C01824=1116.174,356.442,-84.946,-177.177,11.022,149.491
C01825=1116.170,356.689,-84.982,-177.174,11.024,149.491
C01826=1116.166,356.936,-85.017,-177.170,11.027,149.490
C01827=1116.163,357.184,-85.053,-177.167,11.029,149.490
C01828=1116.158,357.431,-85.089,-177.163,11.031,149.490
C01829=1116.155,357.678,-85.125,-177.160,11.034,149.490
C01830=1116.151,357.926,-85.161,-177.157,11.036,149.489
C01831=1116.147,358.173,-85.196,-177.153,11.039,149.489
C01832=1116.143,358.421,-85.232,-177.150,11.041,149.489
C01833=1116.140,358.668,-85.269,-177.146,11.043,149.489
C01834=1116.136,358.916,-85.304,-177.143,11.046,149.488
C01835=1116.132,359.163,-85.340,-177.140,11.048,149.488
C01836=1116.128,359.411,-85.376,-177.136,11.051,149.488
C01837=1116.125,359.658,-85.412,-177.133,11.053,149.487
C01838=1116.121,359.905,-85.448,-177.129,11.055,149.487
C01839=1116.117,360.153,-85.484,-177.126,11.058,149.487
C01840=1116.113,360.400,-85.520,-177.123,11.060,149.487
C01841=1116.110,360.647,-85.556,-177.119,11.063,149.486
C01842=1116.105,360.895,-85.593,-177.116,11.065,149.486
C01843=1116.102,361.142,-85.628,-177.113,11.067,149.486
C01844=1116.098,361.390,-85.664,-177.109,11.070,149.486
C01845=1116.094,361.602,-85.695,-177.107,11.072,149.486
C01846=1116.091,361.813,-85.726,-177.104,11.073,149.485
C01847=1116.089,362.025,-85.757,-177.101,11.076,149.485
C01848=1116.085,362.237,-85.788,-177.098,11.077,149.485
C01849=1116.082,362.449,-85.819,-177.095,11.080,149.485
C01850=1116.078,362.662,-85.850,-177.092,11.082,149.484
C01851=1116.075,362.874,-85.881,-177.090,11.084,149.484
C01852=1116.072,363.085,-85.911,-177.086,11.086,149.484
C01853=1116.068,363.332,-85.948,-177.083,11.088,149.484
C01854=1116.064,363.579,-85.984,-177.079,11.091,149.483
C01855=1116.061,363.828,-86.021,-177.076,11.093,149.483
C01856=1116.057,364.075,-86.057,-177.073,11.096,149.483
C01857=1116.054,364.322,-86.093,-177.069,11.098,149.483
C01858=1116.050,364.569,-86.129,-177.066,11.100,149.482
C01859=1116.046,364.816,-86.166,-177.062,11.103,149.482
C01860=1116.042,365.064,-86.202,-177.059,11.105,149.482
C01861=1116.038,365.311,-86.238,-177.056,11.108,149.482
C01862=1116.034,365.559,-86.274,-177.052,11.110,149.482
C01863=1116.030,365.806,-86.311,-177.049,11.112,149.481
C01864=1116.027,366.053,-86.347,-177.046,11.114,149.481
C01865=1116.022,366.300,-86.384,-177.043,11.116,149.481
C01866=1116.019,366.548,-86.420,-177.040,11.119,149.480
C01867=1116.015,366.795,-86.457,-177.036,11.121,149.480
C01868=1116.012,367.042,-86.493,-177.033,11.124,149.480
C01869=1116.008,367.290,-86.530,-177.029,11.126,149.480
C01870=1116.003,367.537,-86.566,-177.026,11.129,149.479
C01871=1116.000,367.784,-86.603,-177.023,11.131,149.479
C01872=1115.996,368.031,-86.639,-177.019,11.133,149.479
C01873=1115.993,368.278,-86.676,-177.016,11.136,149.479
C01874=1115.989,368.526,-86.713,-177.013,11.138,149.479
C01875=1115.985,368.773,-86.750,-177.009,11.141,149.478
C01876=1115.981,369.021,-86.785,-177.006,11.143,149.478
C01877=1115.977,369.268,-86.822,-177.002,11.146,149.478
C01878=1115.973,369.515,-86.859,-176.999,11.148,149.478
C01879=1115.970,369.762,-86.895,-176.996,11.150,149.477
C01880=1115.966,370.010,-86.932,-176.993,11.153,149.477
C01881=1115.962,370.257,-86.969,-176.989,11.155,149.477
C01882=1115.959,370.504,-87.006,-176.987,11.157,149.477
C01883=1115.955,370.751,-87.042,-176.983,11.160,149.477
C01884=1115.951,370.999,-87.079,-176.980,11.162,149.476
C01885=1115.948,371.246,-87.116,-176.977,11.165,149.476
C01886=1115.944,371.493,-87.153,-176.973,11.167,149.476
C01887=1115.940,371.740,-87.190,-176.970,11.170,149.476
C01888=1115.936,371.988,-87.227,-176.966,11.172,149.475
C01889=1115.933,372.235,-87.263,-176.963,11.174,149.475
C01890=1115.929,372.482,-87.300,-176.960,11.177,149.475
C01891=1115.925,372.730,-87.337,-176.956,11.179,149.475
C01892=1115.921,372.977,-87.374,-176.953,11.182,149.474
C01893=1115.918,373.224,-87.411,-176.950,11.184,149.474
C01894=1115.914,373.471,-87.448,-176.947,11.187,149.474
C01895=1115.910,373.718,-87.485,-176.943,11.189,149.474
C01896=1115.906,373.965,-87.522,-176.940,11.192,149.474
C01897=1115.902,374.213,-87.559,-176.937,11.194,149.473
C01898=1115.898,374.460,-87.596,-176.934,11.197,149.473
C01899=1115.895,374.707,-87.633,-176.930,11.199,149.473
C01900=1115.892,374.955,-87.670,-176.928,11.201,149.473
C01901=1115.888,375.166,-87.702,-176.925,11.203,149.473
C01902=1115.885,375.379,-87.733,-176.922,11.205,149.473
C01903=1115.881,375.590,-87.765,-176.919,11.208,149.473
C01904=1115.879,375.802,-87.797,-176.916,11.210,149.472
C01905=1115.875,376.014,-87.829,-176.914,11.211,149.472
C01906=1115.873,376.226,-87.861,-176.911,11.214,149.472
C01907=1115.868,376.437,-87.893,-176.908,11.216,149.472
C01908=1115.866,376.649,-87.925,-176.905,11.219,149.472
C01909=1115.862,376.896,-87.962,-176.902,11.221,149.472
C01910=1115.858,377.144,-87.999,-176.899,11.223,149.471
C01911=1115.854,377.391,-88.037,-176.896,11.225,149.471
C01912=1115.851,377.638,-88.073,-176.893,11.228,149.471
C01913=1115.847,377.886,-88.110,-176.890,11.231,149.471
C01914=1115.844,378.132,-88.148,-176.886,11.233,149.471
C01915=1115.840,378.379,-88.184,-176.883,11.236,149.471
C01916=1115.836,378.627,-88.222,-176.880,11.238,149.470
C01917=1115.832,378.874,-88.259,-176.877,11.241,149.470
C01918=1115.829,379.120,-88.297,-176.874,11.243,149.470
C01919=1115.825,379.368,-88.334,-176.870,11.246,149.470
C01920=1115.821,379.615,-88.372,-176.867,11.248,149.470
C01921=1115.818,379.863,-88.409,-176.864,11.251,149.470
C01922=1115.814,380.109,-88.446,-176.861,11.254,149.470
C01923=1115.809,380.357,-88.484,-176.858,11.256,149.469
C01924=1115.806,380.604,-88.522,-176.855,11.259,149.469
C01925=1115.802,380.851,-88.559,-176.851,11.261,149.469
C01926=1115.799,381.099,-88.597,-176.848,11.264,149.469
C01927=1115.795,381.345,-88.634,-176.845,11.267,149.469
C01928=1115.791,381.593,-88.671,-176.842,11.269,149.469
C01929=1115.788,381.840,-88.709,-176.839,11.272,149.469
C01930=1115.784,382.087,-88.746,-176.836,11.275,149.468
C01931=1115.780,382.334,-88.784,-176.832,11.277,149.468
C01932=1115.777,382.581,-88.821,-176.829,11.280,149.468
C01933=1115.773,382.829,-88.859,-176.826,11.282,149.468
C01934=1115.769,383.075,-88.897,-176.823,11.285,149.468
C01935=1115.765,383.323,-88.935,-176.820,11.288,149.468
C01936=1115.762,383.569,-88.972,-176.817,11.290,149.468
C01937=1115.758,383.817,-89.009,-176.815,11.293,149.468
C01938=1115.754,384.064,-89.047,-176.813,11.295,149.468
C01939=1115.751,384.311,-89.085,-176.810,11.298,149.468
C01940=1115.747,384.558,-89.123,-176.808,11.300,149.468
C01941=1115.743,384.805,-89.161,-176.806,11.302,149.468
C01942=1115.739,385.052,-89.198,-176.803,11.305,149.468
C01943=1115.736,385.300,-89.236,-176.801,11.307,149.468
C01944=1115.732,385.546,-89.273,-176.798,11.309,149.468
C01945=1115.729,385.793,-89.311,-176.796,11.312,149.468
C01946=1115.725,386.040,-89.350,-176.794,11.314,149.468
C01947=1115.721,386.288,-89.388,-176.791,11.317,149.468
C01948=1115.717,386.535,-89.424,-176.789,11.319,149.468
C01949=1115.714,386.782,-89.462,-176.787,11.321,149.468
C01950=1115.710,387.030,-89.501,-176.784,11.324,149.468
C01951=1115.706,387.276,-89.538,-176.782,11.327,149.468
C01952=1115.703,387.523,-89.576,-176.779,11.330,149.468
C01953=1115.699,387.770,-89.614,-176.778,11.332,149.469
C01954=1115.695,388.018,-89.652,-176.775,11.335,149.469
C01955=1115.692,388.264,-89.690,-176.773,11.337,149.469
C01956=1115.689,388.511,-89.728,-176.770,11.340,149.469
C01957=1115.685,388.724,-89.761,-176.768,11.343,149.469
C01958=1115.682,388.934,-89.793,-176.767,11.345,149.469
C01959=1115.679,389.147,-89.826,-176.765,11.347,149.469
C01960=1115.676,389.358,-89.858,-176.763,11.350,149.469
C01961=1115.673,389.571,-89.891,-176.761,11.352,149.470
C01962=1115.670,389.781,-89.923,-176.759,11.355,149.470
C01963=1115.666,389.994,-89.956,-176.757,11.357,149.470
C01964=1115.664,390.205,-89.988,-176.755,11.359,149.470
C01965=1115.660,390.453,-90.027,-176.753,11.362,149.470
C01966=1115.656,390.699,-90.065,-176.750,11.366,149.470
C01967=1115.653,390.946,-90.102,-176.748,11.368,149.470
C01968=1115.648,391.193,-90.141,-176.746,11.371,149.471
C01969=1115.645,391.441,-90.179,-176.744,11.375,149.471
C01970=1115.642,391.688,-90.217,-176.742,11.377,149.471
C01971=1115.638,391.934,-90.255,-176.739,11.380,149.471
C01972=1115.634,392.181,-90.293,-176.737,11.383,149.472
C01973=1115.631,392.429,-90.332,-176.735,11.386,149.472
C01974=1115.627,392.676,-90.369,-176.733,11.389,149.472
C01975=1115.624,392.923,-90.407,-176.731,11.392,149.472
C01976=1115.620,393.170,-90.447,-176.729,11.396,149.473
C01977=1115.616,393.416,-90.484,-176.726,11.399,149.473
C01978=1115.612,393.664,-90.523,-176.725,11.402,149.473
C01979=1115.609,393.911,-90.561,-176.723,11.405,149.474
C01980=1115.605,394.158,-90.599,-176.720,11.408,149.474
C01981=1115.602,394.405,-90.638,-176.718,11.412,149.474
C01982=1115.598,394.652,-90.676,-176.716,11.415,149.475
C01983=1115.594,394.899,-90.714,-176.714,11.419,149.475
C01984=1115.590,395.146,-90.753,-176.712,11.421,149.475
C01985=1115.587,395.393,-90.791,-176.710,11.425,149.476
C01986=1115.583,395.640,-90.829,-176.708,11.428,149.476
C01987=1115.580,395.887,-90.868,-176.706,11.432,149.476
C01988=1115.576,396.134,-90.906,-176.704,11.435,149.477
C01989=1115.573,396.381,-90.944,-176.702,11.439,149.477
C01990=1115.568,396.628,-90.983,-176.700,11.443,149.478
C01991=1115.565,396.875,-91.021,-176.698,11.446,149.478
C01992=1115.562,397.122,-91.060,-176.696,11.450,149.478
C01993=1115.558,397.369,-91.098,-176.694,11.453,149.479
C01994=1115.554,397.616,-91.136,-176.692,11.457,149.479
C01995=1115.551,397.863,-91.175,-176.690,11.461,149.480
C01996=1115.547,398.110,-91.214,-176.688,11.464,149.480
C01997=1115.543,398.357,-91.252,-176.686,11.468,149.481
C01998=1115.540,398.604,-91.290,-176.684,11.471,149.481
C01999=1115.536,398.851,-91.330,-176.683,11.475,149.482
C02000=1115.533,399.098,-91.368,-176.680,11.480,149.482
C02001=1115.529,399.344,-91.406,-176.678,11.483,149.483
C02002=1115.525,399.592,-91.445,-176.677,11.487,149.483
C02003=1115.522,399.839,-91.484,-176.675,11.491,149.484
C02004=1115.518,400.086,-91.522,-176.673,11.495,149.484
C02005=1115.515,400.333,-91.561,-176.671,11.498,149.485
C02006=1115.511,400.579,-91.600,-176.669,11.503,149.486
C02007=1115.507,400.827,-91.638,-176.667,11.507,149.486
C02008=1115.504,401.073,-91.677,-176.666,11.511,149.487
C02009=1115.500,401.321,-91.715,-176.664,11.515,149.487
C02010=1115.496,401.568,-91.755,-176.662,11.519,149.488
C02011=1115.493,401.814,-91.793,-176.660,11.523,149.489
C02012=1115.489,402.061,-91.831,-176.659,11.527,149.489
C02013=1115.486,402.273,-91.865,-176.657,11.531,149.490
C02014=1115.483,402.484,-91.899,-176.655,11.535,149.490
C02015=1115.480,402.696,-91.932,-176.654,11.538,149.491
C02016=1115.477,402.907,-91.965,-176.653,11.542,149.491
C02017=1115.474,403.119,-91.998,-176.651,11.545,149.492
C02018=1115.471,403.331,-92.031,-176.650,11.550,149.493
C02019=1115.468,403.542,-92.065,-176.648,11.553,149.493
C02020=1115.465,403.754,-92.098,-176.647,11.556,149.494
C02021=1115.461,404.001,-92.137,-176.645,11.561,149.495
C02022=1115.458,404.247,-92.176,-176.643,11.565,149.495
C02023=1115.454,404.494,-92.215,-176.641,11.570,149.496
C02024=1115.450,404.742,-92.253,-176.640,11.574,149.497
C02025=1115.446,404.989,-92.293,-176.638,11.579,149.498
C02026=1115.444,405.235,-92.331,-176.637,11.583,149.498
C02027=1115.440,405.482,-92.370,-176.635,11.588,149.499
C02028=1115.436,405.729,-92.410,-176.634,11.592,149.500
C02029=1115.433,405.976,-92.449,-176.632,11.598,149.501
C02030=1115.429,406.223,-92.488,-176.630,11.603,149.502
C02031=1115.426,406.470,-92.526,-176.629,11.607,149.503
C02032=1115.422,406.717,-92.565,-176.627,11.612,149.503
C02033=1115.418,406.964,-92.604,-176.626,11.616,149.504
C02034=1115.414,407.211,-92.644,-176.624,11.621,149.505
C02035=1115.411,407.457,-92.683,-176.623,11.626,149.506
C02036=1115.407,407.704,-92.722,-176.621,11.631,149.507
C02037=1115.404,407.951,-92.761,-176.620,11.636,149.508
C02038=1115.401,408.198,-92.800,-176.618,11.641,149.509
C02039=1115.397,408.445,-92.839,-176.617,11.646,149.510
C02040=1115.393,408.692,-92.878,-176.615,11.652,149.511
C02041=1115.390,408.939,-92.918,-176.614,11.656,149.512
C02042=1115.386,409.186,-92.957,-176.612,11.661,149.513
C02043=1115.383,409.433,-92.996,-176.611,11.666,149.514
C02044=1115.379,409.680,-93.035,-176.609,11.672,149.515
C02045=1115.376,409.926,-93.075,-176.608,11.677,149.516
C02046=1115.372,410.173,-93.115,-176.607,11.682,149.517
C02047=1115.368,410.420,-93.154,-176.605,11.688,149.518
C02048=1115.366,410.667,-93.193,-176.604,11.693,149.519
C02049=1115.362,410.914,-93.232,-176.602,11.698,149.520
C02050=1115.358,411.161,-93.271,-176.601,11.704,149.521
C02051=1115.355,411.408,-93.310,-176.600,11.710,149.522
C02052=1115.351,411.654,-93.350,-176.598,11.715,149.523
C02053=1115.348,411.901,-93.390,-176.597,11.720,149.524
C02054=1115.344,412.148,-93.429,-176.596,11.726,149.525
C02055=1115.341,412.395,-93.468,-176.595,11.731,149.527
C02056=1115.337,412.641,-93.508,-176.593,11.737,149.528
C02057=1115.334,412.888,-93.547,-176.592,11.742,149.529
C02058=1115.330,413.135,-93.587,-176.591,11.748,149.530
C02059=1115.326,413.382,-93.626,-176.590,11.754,149.531
C02060=1115.324,413.629,-93.666,-176.589,11.759,149.532
C02061=1115.320,413.876,-93.705,-176.587,11.766,149.534
C02062=1115.318,414.123,-93.745,-176.586,11.772,149.535
C02063=1115.316,414.370,-93.784,-176.585,11.777,149.536
C02064=1115.315,414.617,-93.823,-176.584,11.783,149.538
C02065=1115.314,414.864,-93.863,-176.583,11.789,149.539
C02066=1115.313,415.111,-93.902,-176.582,11.795,149.540
C02067=1115.313,415.358,-93.941,-176.581,11.801,149.541
C02068=1115.314,415.604,-93.980,-176.580,11.807,149.543
C02069=1115.316,415.816,-94.014,-176.579,11.813,149.544
C02070=1115.317,416.026,-94.047,-176.578,11.817,149.545
C02071=1115.318,416.239,-94.080,-176.577,11.823,149.546
C02072=1115.321,416.450,-94.113,-176.577,11.828,149.547
C02073=1115.324,416.661,-94.146,-176.576,11.833,149.549
C02074=1115.327,416.872,-94.179,-176.575,11.838,149.550
C02075=1115.330,417.084,-94.212,-176.574,11.844,149.551
C02076=1115.333,417.294,-94.246,-176.574,11.849,149.552
C02077=1114.914,417.294,-94.309,-176.566,11.854,149.551
C02078=1114.911,417.082,-94.275,-176.567,11.848,149.550
C02079=1114.908,416.872,-94.242,-176.568,11.843,149.549
C02080=1114.904,416.660,-94.209,-176.568,11.838,149.548
C02081=1114.902,416.449,-94.175,-176.569,11.832,149.547
C02082=1114.900,416.238,-94.142,-176.570,11.827,149.546
C02083=1114.898,416.026,-94.109,-176.571,11.822,149.544
C02084=1114.896,415.815,-94.076,-176.572,11.816,149.543
C02085=1114.895,415.604,-94.042,-176.573,11.811,149.542
C02086=1114.895,415.357,-94.003,-176.573,11.805,149.541
C02087=1114.894,415.110,-93.964,-176.575,11.799,149.539
C02088=1114.894,414.863,-93.925,-176.576,11.793,149.538
C02089=1114.896,414.617,-93.886,-176.577,11.787,149.537
C02090=1114.896,414.369,-93.846,-176.579,11.781,149.536
C02091=1114.898,414.123,-93.807,-176.580,11.775,149.534
C02092=1114.901,413.875,-93.768,-176.581,11.770,149.533
C02093=1114.904,413.629,-93.728,-176.582,11.764,149.532
C02094=1114.907,413.382,-93.689,-176.583,11.757,149.531
C02095=1114.911,413.135,-93.649,-176.585,11.752,149.529
C02096=1114.914,412.889,-93.609,-176.586,11.746,149.528
C02097=1114.918,412.642,-93.570,-176.587,11.741,149.527
C02098=1114.922,412.395,-93.531,-176.588,11.735,149.526
C02099=1114.925,412.148,-93.492,-176.590,11.729,149.525
C02100=1114.929,411.902,-93.452,-176.591,11.723,149.524
C02101=1114.932,411.654,-93.412,-176.593,11.718,149.523
C02102=1114.935,411.407,-93.373,-176.594,11.713,149.521
C02103=1114.939,411.160,-93.333,-176.595,11.707,149.520
C02104=1114.942,410.914,-93.293,-176.597,11.702,149.519
C02105=1114.946,410.667,-93.254,-176.598,11.696,149.518
C02106=1114.949,410.420,-93.215,-176.600,11.691,149.517
C02107=1114.953,410.173,-93.176,-176.601,11.685,149.516
C02108=1114.957,409.926,-93.136,-176.602,11.680,149.515
C02109=1114.960,409.679,-93.097,-176.604,11.675,149.514
C02110=1114.963,409.432,-93.059,-176.606,11.670,149.513
C02111=1114.967,409.185,-93.019,-176.607,11.665,149.512
C02112=1114.970,408.939,-92.979,-176.609,11.659,149.511
C02113=1114.974,408.692,-92.940,-176.610,11.655,149.510
C02114=1114.977,408.445,-92.901,-176.611,11.650,149.509
C02115=1114.981,408.198,-92.862,-176.613,11.644,149.508
C02116=1114.984,407.951,-92.822,-176.614,11.639,149.507
C02117=1114.989,407.705,-92.783,-176.616,11.634,149.506
C02118=1114.992,407.458,-92.744,-176.617,11.630,149.506
C02119=1114.995,407.211,-92.706,-176.619,11.625,149.505
C02120=1114.999,406.964,-92.666,-176.620,11.619,149.504
C02121=1115.002,406.717,-92.627,-176.622,11.615,149.503
C02122=1115.006,406.470,-92.588,-176.624,11.610,149.502
C02123=1115.010,406.223,-92.549,-176.625,11.605,149.501
C02124=1115.014,405.976,-92.510,-176.627,11.600,149.500
C02125=1115.017,405.729,-92.471,-176.629,11.596,149.500
C02126=1115.020,405.482,-92.432,-176.630,11.591,149.499
C02127=1115.024,405.235,-92.393,-176.632,11.586,149.498
C02128=1115.027,404.988,-92.354,-176.633,11.582,149.497
C02129=1115.031,404.741,-92.314,-176.635,11.577,149.496
C02130=1115.034,404.495,-92.276,-176.637,11.573,149.496
C02131=1115.038,404.248,-92.238,-176.639,11.568,149.495
C02132=1115.042,404.001,-92.198,-176.640,11.564,149.494
C02133=1115.046,403.754,-92.159,-176.642,11.559,149.494
C02134=1115.049,403.542,-92.126,-176.644,11.555,149.493
C02135=1115.051,403.331,-92.093,-176.645,11.551,149.492
C02136=1115.054,403.120,-92.059,-176.647,11.548,149.492
C02137=1115.057,402.908,-92.026,-176.648,11.545,149.491
C02138=1115.060,402.696,-91.992,-176.650,11.541,149.491
C02139=1115.064,402.484,-91.959,-176.651,11.537,149.490
C02140=1115.067,402.273,-91.926,-176.653,11.533,149.489
C02141=1115.070,402.062,-91.893,-176.654,11.530,149.489
C02142=1115.073,401.815,-91.854,-176.656,11.525,149.488
C02143=1115.077,401.568,-91.815,-176.658,11.521,149.488
C02144=1115.080,401.321,-91.777,-176.660,11.518,149.487
C02145=1115.084,401.074,-91.738,-176.662,11.513,149.486
C02146=1115.088,400.826,-91.699,-176.664,11.509,149.486
C02147=1115.091,400.580,-91.661,-176.665,11.505,149.485
C02148=1115.095,400.333,-91.622,-176.668,11.501,149.485
C02149=1115.099,400.086,-91.583,-176.669,11.497,149.484
C02150=1115.102,399.839,-91.545,-176.671,11.493,149.483
C02151=1115.106,399.592,-91.506,-176.673,11.489,149.483
C02152=1115.110,399.345,-91.467,-176.675,11.486,149.483
C02153=1115.113,399.098,-91.429,-176.677,11.481,149.482
C02154=1115.117,398.851,-91.390,-176.679,11.477,149.481
C02155=1115.120,398.604,-91.351,-176.681,11.474,149.481
C02156=1115.124,398.358,-91.313,-176.683,11.470,149.480
C02157=1115.128,398.111,-91.274,-176.685,11.466,149.480
C02158=1115.131,397.863,-91.236,-176.687,11.463,149.480
C02159=1115.135,397.616,-91.197,-176.688,11.459,149.479
C02160=1115.138,397.370,-91.159,-176.691,11.455,149.479
C02161=1115.142,397.122,-91.121,-176.693,11.451,149.478
C02162=1115.145,396.876,-91.082,-176.695,11.447,149.478
C02163=1115.149,396.628,-91.043,-176.697,11.444,149.477
C02164=1115.153,396.382,-91.004,-176.699,11.441,149.477
C02165=1115.156,396.134,-90.967,-176.701,11.437,149.477
C02166=1115.160,395.887,-90.928,-176.703,11.434,149.476
C02167=1115.163,395.640,-90.889,-176.705,11.430,149.476
C02168=1115.168,395.393,-90.851,-176.708,11.427,149.475
C02169=1115.171,395.146,-90.813,-176.710,11.423,149.475
C02170=1115.175,394.899,-90.774,-176.711,11.421,149.475
C02171=1115.178,394.653,-90.736,-176.713,11.417,149.474
C02172=1115.182,394.405,-90.698,-176.715,11.414,149.474
C02173=1115.185,394.158,-90.659,-176.717,11.410,149.474
C02174=1115.190,393.911,-90.621,-176.720,11.407,149.473
C02175=1115.193,393.664,-90.583,-176.722,11.403,149.473
C02176=1115.196,393.417,-90.545,-176.724,11.400,149.473
C02177=1115.200,393.171,-90.506,-176.727,11.397,149.472
C02178=1115.203,392.923,-90.468,-176.728,11.394,149.472
C02179=1115.207,392.676,-90.430,-176.731,11.391,149.472
C02180=1115.211,392.429,-90.392,-176.733,11.388,149.472
C02181=1115.215,392.182,-90.354,-176.735,11.384,149.471
C02182=1115.218,391.934,-90.316,-176.737,11.381,149.471
C02183=1115.222,391.688,-90.277,-176.739,11.379,149.471
C02184=1115.226,391.441,-90.239,-176.742,11.375,149.471
C02185=1115.229,391.194,-90.201,-176.744,11.372,149.471
C02186=1115.233,390.947,-90.163,-176.746,11.370,149.470
C02187=1115.237,390.699,-90.125,-176.748,11.366,149.470
C02188=1115.240,390.453,-90.087,-176.751,11.363,149.470
C02189=1115.244,390.206,-90.049,-176.753,11.361,149.470
C02190=1115.247,389.994,-90.016,-176.755,11.358,149.470
C02191=1115.250,389.781,-89.983,-176.757,11.355,149.469
C02192=1115.253,389.571,-89.951,-176.759,11.353,149.469
C02193=1115.257,389.358,-89.919,-176.761,11.351,149.469
C02194=1115.259,389.147,-89.886,-176.763,11.348,149.469
C02195=1115.263,388.935,-89.854,-176.764,11.346,149.469
C02196=1115.266,388.724,-89.821,-176.766,11.344,149.469
C02197=1115.269,388.512,-89.788,-176.769,11.342,149.469
C02198=1115.273,388.265,-89.751,-176.771,11.338,149.469
C02199=1115.276,388.018,-89.713,-176.773,11.336,149.468
C02200=1115.279,387.771,-89.675,-176.776,11.333,149.468
C02201=1115.284,387.524,-89.637,-176.778,11.331,149.468
C02202=1115.287,387.276,-89.599,-176.780,11.328,149.468
C02203=1115.291,387.030,-89.561,-176.783,11.326,149.468
C02204=1115.294,386.783,-89.523,-176.785,11.323,149.468
C02205=1115.298,386.536,-89.485,-176.787,11.321,149.468
C02206=1115.302,386.288,-89.447,-176.790,11.317,149.468
C02207=1115.305,386.041,-89.409,-176.792,11.315,149.468
C02208=1115.309,385.795,-89.372,-176.795,11.312,149.468
C02209=1115.313,385.546,-89.334,-176.797,11.310,149.468
C02210=1115.317,385.300,-89.296,-176.800,11.307,149.468
C02211=1115.320,385.053,-89.258,-176.802,11.305,149.468
C02212=1115.324,384.806,-89.221,-176.804,11.303,149.468
C02213=1115.327,384.559,-89.183,-176.807,11.300,149.468
C02214=1115.332,384.311,-89.145,-176.809,11.298,149.468
C02215=1115.335,384.064,-89.107,-176.811,11.296,149.468
C02216=1115.339,383.817,-89.070,-176.814,11.293,149.468
C02217=1115.342,383.570,-89.032,-176.816,11.291,149.468
C02218=1115.346,383.324,-88.994,-176.819,11.288,149.468
C02219=1115.349,383.076,-88.957,-176.822,11.286,149.468
C02220=1115.353,382.829,-88.920,-176.826,11.283,149.468
C02221=1115.357,382.581,-88.881,-176.828,11.280,149.468
C02222=1115.361,382.334,-88.844,-176.832,11.278,149.468
C02223=1115.364,382.087,-88.806,-176.835,11.275,149.468
C02224=1115.368,381.840,-88.769,-176.838,11.273,149.469
C02225=1115.372,381.593,-88.732,-176.841,11.270,149.469
C02226=1115.375,381.346,-88.694,-176.844,11.267,149.469
C02227=1115.379,381.099,-88.656,-176.847,11.265,149.469
C02228=1115.382,380.852,-88.619,-176.850,11.262,149.469
C02229=1115.386,380.605,-88.581,-176.854,11.259,149.469
C02230=1115.390,380.357,-88.544,-176.857,11.257,149.469
C02231=1115.394,380.110,-88.507,-176.860,11.254,149.469
C02232=1115.398,379.863,-88.470,-176.863,11.252,149.470
C02233=1115.401,379.616,-88.432,-176.866,11.249,149.470
C02234=1115.405,379.369,-88.395,-176.869,11.246,149.470
C02235=1115.409,379.121,-88.356,-176.873,11.244,149.470
C02236=1115.413,378.874,-88.320,-176.876,11.241,149.470
C02237=1115.417,378.627,-88.282,-176.879,11.239,149.470
C02238=1115.420,378.380,-88.245,-176.882,11.236,149.470
C02239=1115.423,378.133,-88.208,-176.885,11.234,149.471
C02240=1115.427,377.886,-88.171,-176.889,11.231,149.471
C02241=1115.431,377.639,-88.133,-176.892,11.229,149.471
C02242=1115.435,377.392,-88.096,-176.895,11.226,149.471
C02243=1115.438,377.144,-88.059,-176.898,11.223,149.471
C02244=1115.442,376.897,-88.021,-176.901,11.221,149.471
C02245=1115.446,376.650,-87.985,-176.905,11.218,149.472
C02246=1115.449,376.438,-87.953,-176.907,11.217,149.472
C02247=1115.453,376.226,-87.920,-176.910,11.215,149.472
C02248=1115.456,376.014,-87.888,-176.913,11.212,149.472
C02249=1115.459,375.802,-87.857,-176.916,11.210,149.472
C02250=1115.462,375.590,-87.825,-176.919,11.208,149.472
C02251=1115.465,375.379,-87.794,-176.921,11.206,149.473
C02252=1115.468,375.167,-87.762,-176.923,11.204,149.473
C02253=1115.472,374.955,-87.730,-176.927,11.201,149.473
C02254=1115.475,374.708,-87.693,-176.930,11.199,149.473
C02255=1115.479,374.461,-87.656,-176.933,11.196,149.473
C02256=1115.483,374.213,-87.619,-176.937,11.194,149.473
C02257=1115.487,373.967,-87.582,-176.940,11.192,149.474
C02258=1115.490,373.719,-87.544,-176.943,11.189,149.474
C02259=1115.494,373.472,-87.508,-176.947,11.187,149.474
C02260=1115.498,373.225,-87.471,-176.949,11.185,149.474
C02261=1115.501,372.977,-87.434,-176.953,11.182,149.475
C02262=1115.505,372.730,-87.397,-176.956,11.180,149.475
C02263=1115.509,372.483,-87.360,-176.959,11.177,149.475
C02264=1115.512,372.236,-87.323,-176.962,11.175,149.475
C02265=1115.516,371.989,-87.286,-176.966,11.172,149.475
C02266=1115.520,371.741,-87.249,-176.969,11.170,149.476
C02267=1115.524,371.494,-87.212,-176.972,11.168,149.476
C02268=1115.528,371.247,-87.176,-176.976,11.165,149.476
C02269=1115.532,371.000,-87.139,-176.979,11.163,149.476
C02270=1115.535,370.752,-87.102,-176.982,11.160,149.476
C02271=1115.539,370.505,-87.065,-176.986,11.158,149.477
C02272=1115.543,370.258,-87.029,-176.989,11.155,149.477
C02273=1115.547,370.011,-86.992,-176.993,11.153,149.477
C02274=1115.551,369.764,-86.955,-176.996,11.150,149.477
C02275=1115.554,369.516,-86.919,-176.999,11.148,149.478
C02276=1115.558,369.268,-86.882,-177.002,11.146,149.478
C02277=1115.562,369.021,-86.846,-177.006,11.143,149.478
C02278=1115.565,368.774,-86.809,-177.009,11.141,149.478
C02279=1115.569,368.527,-86.773,-177.012,11.138,149.478
C02280=1115.573,368.280,-86.736,-177.015,11.136,149.479
C02281=1115.576,368.032,-86.699,-177.019,11.134,149.479
C02282=1115.580,367.785,-86.662,-177.022,11.132,149.479
C02283=1115.584,367.538,-86.627,-177.025,11.129,149.479
C02284=1115.588,367.290,-86.590,-177.029,11.127,149.480
C02285=1115.592,367.043,-86.553,-177.032,11.124,149.480
C02286=1115.596,366.796,-86.517,-177.035,11.122,149.480
C02287=1115.600,366.549,-86.480,-177.039,11.120,149.481
C02288=1115.603,366.301,-86.444,-177.042,11.117,149.481
C02289=1115.607,366.054,-86.407,-177.045,11.115,149.481
C02290=1115.610,365.807,-86.371,-177.049,11.112,149.481
C02291=1115.615,365.559,-86.335,-177.052,11.110,149.481
C02292=1115.618,365.312,-86.298,-177.055,11.107,149.482
C02293=1115.622,365.065,-86.261,-177.059,11.105,149.482
C02294=1115.626,364.817,-86.226,-177.062,11.103,149.482
C02295=1115.630,364.570,-86.189,-177.066,11.100,149.482
C02296=1115.633,364.323,-86.154,-177.069,11.098,149.483
C02297=1115.638,364.076,-86.117,-177.072,11.095,149.483
C02298=1115.641,363.829,-86.080,-177.076,11.093,149.483
C02299=1115.645,363.581,-86.044,-177.079,11.091,149.483
C02300=1115.648,363.333,-86.008,-177.083,11.088,149.484
C02301=1115.652,363.086,-85.971,-177.086,11.086,149.484
C02302=1115.655,362.875,-85.940,-177.089,11.084,149.484
C02303=1115.659,362.663,-85.910,-177.091,11.082,149.484
C02304=1115.662,362.450,-85.878,-177.095,11.080,149.485
C02305=1115.665,362.238,-85.847,-177.097,11.078,149.485
C02306=1115.668,362.026,-85.817,-177.101,11.076,149.485
C02307=1115.672,361.814,-85.786,-177.103,11.074,149.485
C02308=1115.675,361.602,-85.755,-177.106,11.072,149.486
C02309=1115.679,361.390,-85.724,-177.109,11.070,149.486
C02310=1115.682,361.143,-85.688,-177.113,11.067,149.486
C02311=1115.686,360.895,-85.652,-177.116,11.065,149.486
C02312=1115.690,360.648,-85.615,-177.119,11.063,149.486
C02313=1115.693,360.401,-85.580,-177.122,11.060,149.487
C02314=1115.697,360.153,-85.544,-177.126,11.058,149.487
C02315=1115.701,359.906,-85.507,-177.129,11.055,149.487
C02316=1115.705,359.659,-85.472,-177.133,11.053,149.487
C02317=1115.709,359.411,-85.436,-177.136,11.050,149.488
C02318=1115.712,359.164,-85.400,-177.139,11.048,149.488
C02319=1115.716,358.916,-85.364,-177.143,11.046,149.488
C02320=1115.720,358.669,-85.328,-177.146,11.043,149.489
C02321=1115.723,358.422,-85.292,-177.150,11.041,149.489
C02322=1115.727,358.174,-85.256,-177.153,11.038,149.489
C02323=1115.731,357.927,-85.220,-177.156,11.036,149.489
C02324=1115.735,357.679,-85.185,-177.160,11.034,149.490
C02325=1115.739,357.432,-85.150,-177.163,11.031,149.490
C02326=1115.743,357.186,-85.113,-177.167,11.029,149.490
C02327=1115.747,356.938,-85.077,-177.170,11.026,149.490
C02328=1115.751,356.690,-85.042,-177.173,11.024,149.490
C02329=1115.754,356.443,-85.006,-177.177,11.022,149.491
C02330=1115.758,356.195,-84.971,-177.180,11.019,149.491
C02331=1115.762,355.948,-84.935,-177.184,11.017,149.491
C02332=1115.766,355.700,-84.899,-177.187,11.014,149.492
C02333=1115.769,355.453,-84.863,-177.190,11.012,149.492
C02334=1115.773,355.205,-84.827,-177.193,11.010,149.492
C02335=1115.777,354.959,-84.792,-177.197,11.007,149.492
C02336=1115.781,354.711,-84.756,-177.200,11.005,149.493
C02337=1115.785,354.464,-84.721,-177.204,11.002,149.493
C02338=1115.788,354.216,-84.685,-177.207,11.000,149.493
C02339=1115.792,353.969,-84.650,-177.210,10.998,149.493
C02340=1115.796,353.721,-84.614,-177.214,10.995,149.493
C02341=1115.801,353.474,-84.578,-177.218,10.992,149.494
C02342=1115.804,353.227,-84.543,-177.221,10.990,149.494
C02343=1115.808,352.979,-84.507,-177.225,10.987,149.494
C02344=1115.812,352.731,-84.472,-177.228,10.985,149.495
C02345=1115.816,352.483,-84.437,-177.231,10.982,149.495
C02346=1115.819,352.236,-84.401,-177.235,10.980,149.495
C02347=1115.824,351.989,-84.366,-177.238,10.977,149.495
C02348=1115.827,351.742,-84.331,-177.241,10.975,149.495
C02349=1115.831,351.494,-84.295,-177.245,10.972,149.496
C02350=1115.835,351.247,-84.260,-177.248,10.970,149.496
C02351=1115.839,350.999,-84.225,-177.251,10.968,149.496
C02352=1115.843,350.752,-84.189,-177.254,10.965,149.496
C02353=1115.846,350.504,-84.154,-177.258,10.962,149.496
C02354=1115.850,350.257,-84.118,-177.262,10.960,149.497
C02355=1115.855,350.009,-84.084,-177.265,10.957,149.497
C02356=1115.858,349.762,-84.048,-177.269,10.955,149.497
C02357=1115.862,349.514,-84.013,-177.272,10.952,149.498
C02358=1115.865,349.302,-83.983,-177.274,10.950,149.498
C02359=1115.869,349.090,-83.952,-177.278,10.948,149.498
C02360=1115.872,348.878,-83.923,-177.280,10.946,149.498
C02361=1115.875,348.666,-83.892,-177.283,10.943,149.498
C02362=1115.879,348.454,-83.862,-177.286,10.942,149.498
C02363=1115.882,348.241,-83.833,-177.288,10.940,149.499
C02364=1115.886,348.029,-83.802,-177.291,10.937,149.499
C02365=1115.889,347.817,-83.772,-177.294,10.935,149.499
C02366=1115.893,347.570,-83.737,-177.297,10.933,149.499
C02367=1115.897,347.322,-83.702,-177.300,10.930,149.499
C02368=1115.900,347.075,-83.667,-177.304,10.928,149.500
C02369=1115.904,346.828,-83.632,-177.307,10.925,149.500
C02370=1115.908,346.579,-83.597,-177.310,10.923,149.500
C02371=1115.912,346.333,-83.562,-177.313,10.921,149.500
C02372=1115.916,346.085,-83.527,-177.316,10.918,149.500
C02373=1115.920,345.837,-83.491,-177.319,10.916,149.501
C02374=1115.924,345.590,-83.457,-177.323,10.914,149.501
C02375=1115.927,345.342,-83.422,-177.326,10.911,149.501
C02376=1115.931,345.094,-83.387,-177.329,10.908,149.501
C02377=1115.936,344.847,-83.352,-177.332,10.906,149.501
C02378=1115.939,344.599,-83.317,-177.335,10.903,149.501
C02379=1115.944,344.352,-83.282,-177.339,10.901,149.502
C02380=1115.947,344.105,-83.248,-177.342,10.898,149.502
C02381=1115.951,343.857,-83.213,-177.345,10.896,149.502
C02382=1115.955,343.609,-83.178,-177.348,10.893,149.502
C02383=1115.959,343.362,-83.143,-177.351,10.892,149.502
C02384=1115.963,343.115,-83.109,-177.354,10.889,149.503
C02385=1115.967,342.867,-83.074,-177.358,10.887,149.503
C02386=1115.971,342.619,-83.038,-177.361,10.884,149.503
C02387=1115.974,342.372,-83.005,-177.364,10.881,149.503
C02388=1115.978,342.124,-82.970,-177.367,10.879,149.503
C02389=1115.983,341.877,-82.935,-177.370,10.876,149.504
C02390=1115.987,341.629,-82.900,-177.374,10.874,149.504
C02391=1115.990,341.382,-82.866,-177.377,10.872,149.504
C02392=1115.994,341.134,-82.831,-177.380,10.869,149.504
C02393=1115.999,340.886,-82.797,-177.383,10.866,149.504
C02394=1116.002,340.639,-82.762,-177.387,10.864,149.505
C02395=1116.006,340.391,-82.727,-177.389,10.862,149.505
C02396=1116.010,340.144,-82.692,-177.392,10.859,149.505
C02397=1116.014,339.896,-82.658,-177.396,10.857,149.505
C02398=1116.018,339.648,-82.624,-177.399,10.854,149.505
C02399=1116.021,339.400,-82.589,-177.402,10.852,149.506
C02400=1116.026,339.154,-82.554,-177.405,10.850,149.506
C02401=1116.030,338.906,-82.519,-177.408,10.847,149.506
C02402=1116.034,338.658,-82.485,-177.412,10.844,149.506
C02403=1116.038,338.411,-82.451,-177.415,10.842,149.506
C02404=1116.041,338.163,-82.417,-177.418,10.839,149.507
C02405=1116.046,337.916,-82.382,-177.421,10.837,149.507
C02406=1116.049,337.668,-82.348,-177.425,10.834,149.507
C02407=1116.054,337.421,-82.314,-177.427,10.833,149.507
C02408=1116.057,337.173,-82.279,-177.431,10.830,149.507
C02409=1116.061,336.925,-82.245,-177.433,10.827,149.508
C02410=1116.065,336.678,-82.211,-177.437,10.825,149.508
C02411=1116.069,336.430,-82.176,-177.440,10.822,149.508
C02412=1116.073,336.182,-82.142,-177.443,10.820,149.508
C02413=1116.077,335.935,-82.107,-177.446,10.817,149.508
C02414=1116.081,335.722,-82.079,-177.449,10.815,149.509
C02415=1116.084,335.510,-82.049,-177.452,10.813,149.509
C02416=1116.087,335.297,-82.019,-177.455,10.811,149.509
C02417=1116.091,335.086,-81.990,-177.457,10.809,149.509
C02418=1116.094,334.873,-81.961,-177.460,10.807,149.509
C02419=1116.098,334.661,-81.932,-177.463,10.805,149.509
C02420=1116.101,334.449,-81.902,-177.465,10.803,149.510
C02421=1116.103,334.237,-81.873,-177.468,10.800,149.510
C02422=1116.108,333.989,-81.839,-177.471,10.798,149.510
C02423=1116.112,333.741,-81.805,-177.475,10.795,149.510
C02424=1116.116,333.493,-81.771,-177.478,10.792,149.510
C02425=1116.120,333.246,-81.737,-177.481,10.790,149.510
C02426=1116.123,332.998,-81.703,-177.484,10.788,149.511
C02427=1116.128,332.750,-81.669,-177.487,10.786,149.511
C02428=1116.132,332.503,-81.635,-177.490,10.783,149.511
C02429=1116.135,332.255,-81.601,-177.493,10.781,149.511
C02430=1116.140,332.007,-81.567,-177.497,10.778,149.511
C02431=1116.144,331.760,-81.533,-177.500,10.776,149.512
C02432=1116.147,331.513,-81.499,-177.503,10.773,149.512
C02433=1116.152,331.264,-81.465,-177.506,10.770,149.512
C02434=1116.155,331.017,-81.431,-177.509,10.768,149.512
C02435=1116.159,330.770,-81.397,-177.512,10.765,149.512
C02436=1116.164,330.522,-81.363,-177.516,10.763,149.512
C02437=1116.168,330.274,-81.329,-177.519,10.760,149.513
C02438=1116.171,330.026,-81.296,-177.521,10.758,149.513
C02439=1116.175,329.779,-81.262,-177.525,10.756,149.513
C02440=1116.179,329.531,-81.227,-177.528,10.753,149.513
C02441=1116.183,329.283,-81.194,-177.531,10.751,149.514
C02442=1116.187,329.036,-81.160,-177.534,10.748,149.514
C02443=1116.191,328.788,-81.127,-177.538,10.746,149.514
C02444=1116.194,328.540,-81.093,-177.541,10.743,149.514
C02445=1116.199,328.292,-81.059,-177.544,10.741,149.514
C02446=1116.203,328.045,-81.025,-177.547,10.738,149.514
C02447=1116.207,327.797,-80.992,-177.550,10.736,149.515
C02448=1116.210,327.550,-80.958,-177.553,10.733,149.515
C02449=1116.214,327.302,-80.924,-177.556,10.731,149.515
C02450=1116.219,327.054,-80.891,-177.559,10.729,149.515
C02451=1116.223,326.807,-80.857,-177.562,10.726,149.515
C02452=1116.227,326.558,-80.823,-177.566,10.723,149.516
C02453=1116.231,326.311,-80.789,-177.569,10.721,149.516
C02454=1116.235,326.064,-80.756,-177.572,10.718,149.516
C02455=1116.239,325.816,-80.723,-177.575,10.716,149.516
C02456=1116.243,325.569,-80.689,-177.578,10.713,149.516
C02457=1116.246,325.320,-80.656,-177.581,10.711,149.516
C02458=1116.250,325.073,-80.623,-177.585,10.708,149.517
C02459=1116.255,324.824,-80.589,-177.588,10.706,149.517
C02460=1116.259,324.577,-80.555,-177.591,10.703,149.517
C02461=1116.263,324.329,-80.521,-177.594,10.701,149.517
C02462=1116.267,324.081,-80.488,-177.597,10.699,149.517
C02463=1116.271,323.833,-80.455,-177.600,10.696,149.518
C02464=1116.275,323.586,-80.421,-177.603,10.694,149.518
C02465=1116.279,323.339,-80.388,-177.607,10.691,149.518
C02466=1116.283,323.091,-80.355,-177.609,10.688,149.518
C02467=1116.286,322.842,-80.321,-177.613,10.686,149.518
C02468=1116.291,322.595,-80.288,-177.616,10.683,149.519
C02469=1116.294,322.348,-80.254,-177.619,10.681,149.519
C02470=1116.297,322.135,-80.226,-177.622,10.679,149.519
C02471=1116.301,321.923,-80.198,-177.624,10.677,149.519
C02472=1116.304,321.710,-80.169,-177.627,10.674,149.519
C02473=1116.308,321.498,-80.141,-177.630,10.673,149.519
C02474=1116.311,321.286,-80.113,-177.633,10.670,149.519
C02475=1116.315,321.073,-80.084,-177.635,10.668,149.520
C02476=1116.319,320.861,-80.055,-177.638,10.666,149.520
C02477=1116.321,320.648,-80.027,-177.640,10.663,149.520
C02478=1116.326,320.400,-79.994,-177.644,10.661,149.520
C02479=1116.330,320.153,-79.961,-177.647,10.659,149.520
C02480=1116.334,319.905,-79.927,-177.649,10.656,149.520
C02481=1116.338,319.657,-79.894,-177.653,10.654,149.521
C02482=1116.342,319.409,-79.861,-177.656,10.652,149.521
C02483=1116.346,319.162,-79.828,-177.659,10.649,149.521
C02484=1116.350,318.914,-79.795,-177.662,10.646,149.521
C02485=1116.354,318.667,-79.762,-177.665,10.644,149.521
C02486=1116.357,318.418,-79.729,-177.669,10.641,149.522
C02487=1116.361,318.170,-79.696,-177.672,10.639,149.522
C02488=1116.366,317.923,-79.662,-177.675,10.636,149.522
C02489=1116.369,317.675,-79.630,-177.678,10.633,149.522
C02490=1116.373,317.427,-79.597,-177.680,10.631,149.522
C02491=1116.378,317.179,-79.564,-177.684,10.629,149.523
C02492=1116.382,316.931,-79.531,-177.687,10.627,149.523
C02493=1116.386,316.684,-79.498,-177.690,10.624,149.523
C02494=1116.389,316.436,-79.465,-177.693,10.621,149.523
C02495=1116.393,316.189,-79.432,-177.696,10.619,149.523
C02496=1116.398,315.940,-79.400,-177.700,10.616,149.523
C02497=1116.402,315.692,-79.367,-177.703,10.614,149.524
C02498=1116.405,315.445,-79.334,-177.706,10.611,149.524
C02499=1116.410,315.197,-79.301,-177.709,10.609,149.524
C02500=1116.414,314.949,-79.268,-177.712,10.606,149.524
C02501=1116.417,314.702,-79.236,-177.715,10.603,149.524
C02502=1116.422,314.454,-79.203,-177.718,10.602,149.525
C02503=1116.426,314.205,-79.170,-177.721,10.599,149.525
C02504=1116.430,313.958,-79.137,-177.724,10.596,149.525
C02505=1116.434,313.710,-79.105,-177.727,10.594,149.525
C02506=1116.438,313.462,-79.072,-177.731,10.591,149.525
C02507=1116.442,313.214,-79.039,-177.734,10.589,149.526
C02508=1116.445,312.967,-79.006,-177.737,10.586,149.526
C02509=1116.450,312.718,-78.974,-177.740,10.584,149.526
C02510=1116.453,312.471,-78.941,-177.743,10.581,149.526
C02511=1116.458,312.223,-78.909,-177.747,10.578,149.526
C02512=1116.463,311.976,-78.876,-177.749,10.576,149.526
C02513=1116.466,311.728,-78.844,-177.752,10.574,149.527
C02514=1116.470,311.480,-78.811,-177.755,10.572,149.527
C02515=1116.475,311.232,-78.779,-177.758,10.569,149.527
C02516=1116.478,310.984,-78.746,-177.762,10.566,149.527
C02517=1116.483,310.736,-78.714,-177.765,10.564,149.527
C02518=1116.486,310.488,-78.681,-177.768,10.561,149.527
C02519=1116.490,310.240,-78.649,-177.771,10.558,149.528
C02520=1116.494,309.993,-78.616,-177.774,10.556,149.528
C02521=1116.498,309.744,-78.584,-177.777,10.553,149.528
C02522=1116.502,309.498,-78.552,-177.780,10.551,149.528
C02523=1116.507,309.249,-78.519,-177.784,10.548,149.528
C02524=1116.511,309.001,-78.487,-177.786,10.546,149.528
C02525=1116.515,308.753,-78.454,-177.789,10.544,149.529
C02526=1116.518,308.541,-78.427,-177.792,10.541,149.529
C02527=1116.521,308.328,-78.399,-177.795,10.539,149.529
C02528=1116.526,308.116,-78.371,-177.797,10.537,149.529
C02529=1116.529,307.903,-78.344,-177.800,10.535,149.529
C02530=1116.532,307.690,-78.315,-177.803,10.533,149.529
C02531=1116.536,307.478,-78.288,-177.805,10.531,149.530
C02532=1116.539,307.265,-78.260,-177.808,10.528,149.530
C02533=1116.542,307.053,-78.233,-177.811,10.526,149.530
C02534=1116.547,306.805,-78.200,-177.814,10.524,149.530
C02535=1116.551,306.557,-78.169,-177.817,10.521,149.530
C02536=1116.555,306.309,-78.136,-177.820,10.519,149.530
C02537=1116.559,306.062,-78.104,-177.823,10.516,149.530
C02538=1116.563,305.813,-78.071,-177.826,10.513,149.531
C02539=1116.567,305.565,-78.039,-177.830,10.511,149.531
C02540=1116.571,305.318,-78.008,-177.832,10.509,149.531
C02541=1116.576,305.069,-77.975,-177.835,10.506,149.531
C02542=1116.579,304.821,-77.944,-177.838,10.504,149.531
C02543=1116.583,304.574,-77.910,-177.842,10.501,149.532
C02544=1116.588,304.326,-77.879,-177.845,10.499,149.532
C02545=1116.592,304.078,-77.847,-177.848,10.496,149.532
C02546=1116.596,303.830,-77.815,-177.851,10.493,149.532
C02547=1116.600,303.582,-77.783,-177.854,10.491,149.532
C02548=1116.604,303.335,-77.751,-177.857,10.488,149.532
C02549=1116.608,303.086,-77.719,-177.860,10.486,149.533
C02550=1116.612,302.838,-77.687,-177.863,10.483,149.533
C02551=1116.616,302.591,-77.656,-177.866,10.481,149.533
C02552=1116.621,302.342,-77.623,-177.869,10.478,149.533
C02553=1116.625,302.094,-77.591,-177.872,10.476,149.533
C02554=1116.628,301.846,-77.559,-177.875,10.473,149.534
C02555=1116.633,301.599,-77.528,-177.879,10.471,149.534
C02556=1116.637,301.351,-77.496,-177.881,10.468,149.534
C02557=1116.641,301.103,-77.464,-177.885,10.466,149.534
C02558=1116.645,300.855,-77.432,-177.888,10.463,149.534
C02559=1116.649,300.607,-77.400,-177.891,10.460,149.535
C02560=1116.653,300.359,-77.368,-177.894,10.458,149.535
C02561=1116.658,300.112,-77.336,-177.897,10.456,149.535
C02562=1116.662,299.863,-77.305,-177.900,10.453,149.535
C02563=1116.665,299.615,-77.273,-177.903,10.451,149.535
C02564=1116.670,299.368,-77.242,-177.906,10.448,149.535
C02565=1116.674,299.119,-77.210,-177.909,10.446,149.536
C02566=1116.678,298.871,-77.178,-177.912,10.443,149.536
C02567=1116.682,298.624,-77.146,-177.915,10.440,149.536
C02568=1116.686,298.375,-77.115,-177.918,10.438,149.536
C02569=1116.690,298.128,-77.084,-177.922,10.435,149.536
C02570=1116.694,297.880,-77.052,-177.925,10.432,149.536
C02571=1116.698,297.632,-77.020,-177.927,10.431,149.537
C02572=1116.703,297.384,-76.989,-177.930,10.428,149.537
C02573=1116.707,297.135,-76.957,-177.934,10.426,149.537
C02574=1116.711,296.888,-76.925,-177.937,10.423,149.537
C02575=1116.715,296.639,-76.894,-177.940,10.420,149.537
C02576=1116.719,296.391,-76.862,-177.943,10.418,149.537
C02577=1116.723,296.144,-76.831,-177.946,10.415,149.538
C02578=1116.727,295.895,-76.800,-177.949,10.412,149.538
C02579=1116.731,295.648,-76.768,-177.952,10.410,149.538
C02580=1116.735,295.400,-76.736,-177.955,10.407,149.538
C02581=1116.740,295.152,-76.706,-177.958,10.406,149.538
C02582=1116.743,294.939,-76.678,-177.961,10.403,149.539
C02583=1116.747,294.726,-76.651,-177.963,10.401,149.539
C02584=1116.750,294.514,-76.625,-177.966,10.399,149.539
C02585=1116.753,294.301,-76.598,-177.969,10.396,149.539
C02586=1116.757,294.089,-76.570,-177.971,10.394,149.539
C02587=1116.761,293.876,-76.544,-177.974,10.392,149.539
C02588=1116.764,293.663,-76.517,-177.977,10.390,149.539
C02589=1116.767,293.450,-76.490,-177.979,10.388,149.540
C02590=1116.772,293.202,-76.459,-177.982,10.385,149.540
C02591=1116.776,292.954,-76.427,-177.985,10.383,149.540
C02592=1116.780,292.706,-76.396,-177.988,10.380,149.540
C02593=1116.784,292.458,-76.365,-177.992,10.378,149.540
C02594=1116.788,292.210,-76.334,-177.995,10.375,149.540
C02595=1116.792,291.962,-76.303,-177.998,10.372,149.541
C02596=1116.797,291.714,-76.271,-178.000,10.370,149.541
C02597=1116.801,291.466,-76.240,-178.003,10.368,149.541
C02598=1116.804,291.219,-76.209,-178.007,10.365,149.541
C02599=1116.808,290.970,-76.178,-178.010,10.363,149.541
C02600=1116.813,290.722,-76.147,-178.013,10.360,149.542
C02601=1116.817,290.474,-76.115,-178.016,10.357,149.542
C02602=1116.821,290.226,-76.085,-178.019,10.355,149.542
C02603=1116.825,289.977,-76.054,-178.022,10.352,149.542
C02604=1116.829,289.730,-76.023,-178.025,10.350,149.542
C02605=1116.833,289.482,-75.992,-178.028,10.348,149.542
C02606=1116.838,289.234,-75.961,-178.031,10.345,149.542
C02607=1116.842,288.986,-75.930,-178.034,10.343,149.543
C02608=1116.846,288.738,-75.898,-178.037,10.340,149.543
C02609=1116.850,288.490,-75.867,-178.040,10.337,149.543
C02610=1116.854,288.241,-75.837,-178.043,10.335,149.543
C02611=1116.858,287.993,-75.806,-178.047,10.332,149.543
C02612=1116.863,287.746,-75.775,-178.049,10.329,149.544
C02613=1116.867,287.497,-75.744,-178.053,10.327,149.544
C02614=1116.871,287.250,-75.713,-178.056,10.324,149.544
C02615=1116.875,287.001,-75.682,-178.058,10.322,149.544
C02616=1116.879,286.753,-75.651,-178.061,10.320,149.544
C02617=1116.884,286.505,-75.621,-178.064,10.317,149.544
C02618=1116.887,286.257,-75.590,-178.068,10.315,149.545
C02619=1116.891,286.009,-75.559,-178.071,10.312,149.545
C02620=1116.896,285.762,-75.528,-178.074,10.309,149.545
C02621=1116.899,285.513,-75.497,-178.077,10.307,149.545
C02622=1116.904,285.265,-75.467,-178.080,10.304,149.545
C02623=1116.908,285.017,-75.436,-178.083,10.302,149.546
C02624=1116.912,284.769,-75.405,-178.085,10.300,149.546
C02625=1116.916,284.521,-75.375,-178.089,10.297,149.546
C02626=1116.921,284.273,-75.344,-178.092,10.294,149.546
C02627=1116.924,284.025,-75.313,-178.095,10.292,149.546
C02628=1116.929,283.777,-75.282,-178.098,10.289,149.546
C02629=1116.933,283.529,-75.252,-178.101,10.286,149.546
C02630=1116.937,283.280,-75.221,-178.104,10.284,149.547
C02631=1116.941,283.032,-75.190,-178.107,10.281,149.547
C02632=1116.946,282.784,-75.161,-178.110,10.280,149.547
C02633=1116.950,282.536,-75.130,-178.113,10.277,149.547
C02634=1116.954,282.288,-75.099,-178.116,10.274,149.547
C02635=1116.958,282.040,-75.069,-178.119,10.272,149.548
C02636=1116.963,281.792,-75.038,-178.122,10.269,149.548
C02637=1116.966,281.544,-75.008,-178.125,10.266,149.548
C02638=1116.971,281.331,-74.981,-178.128,10.264,149.548
C02639=1116.974,281.118,-74.956,-178.131,10.262,149.548
C02640=1116.977,280.906,-74.930,-178.133,10.260,149.549
C02641=1116.981,280.693,-74.903,-178.136,10.257,149.549
C02642=1116.984,280.480,-74.877,-178.139,10.255,149.549
C02643=1116.988,280.267,-74.851,-178.142,10.253,149.549
C02644=1116.992,280.054,-74.825,-178.145,10.250,149.549
C02645=1116.995,279.841,-74.799,-178.147,10.248,149.549
C02646=1117.000,279.592,-74.769,-178.150,10.245,149.549
C02647=1117.004,279.345,-74.739,-178.154,10.243,149.550
C02648=1117.008,279.096,-74.708,-178.156,10.240,149.550
C02649=1117.011,278.848,-74.677,-178.160,10.238,149.550
C02650=1117.016,278.600,-74.647,-178.163,10.235,149.550
C02651=1117.020,278.352,-74.617,-178.166,10.232,149.550
C02652=1117.024,278.105,-74.587,-178.169,10.230,149.550
C02653=1117.028,277.855,-74.557,-178.172,10.227,149.551
C02654=1117.032,277.608,-74.527,-178.175,10.224,149.551
C02655=1117.037,277.359,-74.496,-178.178,10.222,149.551
C02656=1117.041,277.111,-74.466,-178.181,10.219,149.551
C02657=1117.045,276.864,-74.436,-178.185,10.216,149.551
C02658=1117.050,276.615,-74.406,-178.188,10.213,149.551
C02659=1117.053,276.367,-74.376,-178.190,10.211,149.552
C02660=1117.057,276.119,-74.346,-178.193,10.208,149.552
C02661=1117.062,275.871,-74.315,-178.196,10.206,149.552
C02662=1117.066,275.622,-74.286,-178.199,10.203,149.552
C02663=1117.070,275.375,-74.256,-178.203,10.201,149.552
C02664=1117.075,275.126,-74.226,-178.205,10.198,149.552
C02665=1117.079,274.879,-74.195,-178.208,10.195,149.552
C02666=1117.083,274.630,-74.166,-178.211,10.192,149.552
C02667=1117.087,274.381,-74.136,-178.214,10.189,149.552
C02668=1117.091,274.133,-74.105,-178.217,10.187,149.553
C02669=1117.095,273.885,-74.076,-178.221,10.184,149.553
C02670=1117.099,273.637,-74.046,-178.224,10.182,149.553
C02671=1117.104,273.389,-74.016,-178.226,10.179,149.553
C02672=1117.108,273.141,-73.986,-178.229,10.176,149.553
C02673=1117.112,272.893,-73.956,-178.232,10.173,149.553
C02674=1117.116,272.645,-73.927,-178.235,10.171,149.553
C02675=1117.121,272.396,-73.897,-178.238,10.169,149.553
C02676=1117.125,272.148,-73.866,-178.240,10.166,149.554
C02677=1117.129,271.900,-73.837,-178.243,10.163,149.554
C02678=1117.134,271.652,-73.808,-178.246,10.160,149.554
C02679=1117.137,271.404,-73.777,-178.249,10.157,149.554
C02680=1117.142,271.156,-73.748,-178.252,10.155,149.554
C02681=1117.146,270.907,-73.718,-178.255,10.153,149.554
C02682=1117.150,270.658,-73.688,-178.257,10.150,149.554
C02683=1117.154,270.411,-73.658,-178.261,10.148,149.554
C02684=1117.158,270.163,-73.628,-178.264,10.145,149.555
C02685=1117.162,269.914,-73.599,-178.267,10.142,149.555
C02686=1117.167,269.666,-73.570,-178.269,10.140,149.555
C02687=1117.171,269.418,-73.540,-178.272,10.137,149.555
C02688=1117.175,269.169,-73.511,-178.275,10.135,149.555
C02689=1117.180,268.921,-73.480,-178.278,10.132,149.555
C02690=1117.184,268.673,-73.450,-178.280,10.130,149.555
C02691=1117.188,268.425,-73.421,-178.283,10.127,149.555
C02692=1117.193,268.177,-73.392,-178.286,10.124,149.555
C02693=1117.197,267.929,-73.362,-178.288,10.122,149.556
C02694=1117.200,267.716,-73.337,-178.291,10.119,149.555
C02695=1117.204,267.503,-73.311,-178.293,10.117,149.556
C02696=1117.207,267.289,-73.286,-178.295,10.115,149.556
C02697=1117.211,267.077,-73.261,-178.298,10.113,149.556
C02698=1117.215,266.864,-73.235,-178.300,10.111,149.556
C02699=1117.218,266.651,-73.210,-178.302,10.109,149.556
C02700=1117.222,266.438,-73.185,-178.305,10.107,149.556
C02701=1117.226,266.225,-73.160,-178.307,10.104,149.556
C02702=1117.230,265.977,-73.130,-178.310,10.102,149.556
C02703=1117.234,265.729,-73.101,-178.312,10.099,149.556
C02704=1117.239,265.480,-73.072,-178.315,10.097,149.556
C02705=1117.243,265.231,-73.042,-178.318,10.095,149.557
C02706=1117.247,264.983,-73.013,-178.321,10.092,149.557
C02707=1117.251,264.735,-72.984,-178.323,10.090,149.557
C02708=1117.256,264.487,-72.954,-178.326,10.087,149.557
C02709=1117.260,264.239,-72.925,-178.329,10.085,149.557
C02710=1117.264,263.991,-72.896,-178.332,10.082,149.557
C02711=1117.268,263.742,-72.866,-178.336,10.079,149.558
C02712=1117.272,263.495,-72.837,-178.339,10.076,149.558
C02713=1117.276,263.246,-72.808,-178.342,10.074,149.558
C02714=1117.281,262.997,-72.779,-178.345,10.071,149.558
C02715=1117.285,262.749,-72.750,-178.349,10.067,149.558
C02716=1117.289,262.502,-72.721,-178.352,10.065,149.558
C02717=1117.294,262.253,-72.691,-178.355,10.062,149.559
C02718=1117.298,262.004,-72.662,-178.358,10.060,149.559
C02719=1117.302,261.756,-72.633,-178.362,10.056,149.559
C02720=1117.306,261.508,-72.604,-178.365,10.053,149.559
C02721=1117.310,261.260,-72.575,-178.368,10.050,149.559
C02722=1117.315,261.012,-72.546,-178.371,10.048,149.559
C02723=1117.319,260.763,-72.517,-178.374,10.045,149.559
C02724=1117.323,260.515,-72.487,-178.377,10.043,149.560
C02725=1117.328,260.266,-72.459,-178.380,10.039,149.560
C02726=1117.331,260.018,-72.430,-178.383,10.036,149.560
C02727=1117.336,259.771,-72.401,-178.386,10.033,149.560
C02728=1117.341,259.522,-72.372,-178.389,10.031,149.560
C02729=1117.345,259.274,-72.342,-178.392,10.028,149.560
C02730=1117.349,259.025,-72.314,-178.395,10.025,149.560
C02731=1117.353,258.777,-72.285,-178.398,10.022,149.560
C02732=1117.357,258.529,-72.256,-178.401,10.019,149.560
C02733=1117.361,258.281,-72.228,-178.404,10.017,149.560
C02734=1117.365,258.032,-72.198,-178.407,10.014,149.560
C02735=1117.371,257.784,-72.170,-178.409,10.011,149.560
C02736=1117.375,257.536,-72.140,-178.412,10.008,149.561
C02737=1117.378,257.287,-72.112,-178.415,10.006,149.561
C02738=1117.383,257.039,-72.083,-178.418,10.002,149.561
C02739=1117.388,256.791,-72.054,-178.421,10.000,149.561
C02740=1117.391,256.543,-72.025,-178.424,9.997,149.561
C02741=1117.396,256.294,-71.997,-178.427,9.994,149.561
C02742=1117.400,256.045,-71.968,-178.429,9.991,149.561
C02743=1117.404,255.798,-71.940,-178.430,9.990,149.561
C02744=1117.409,255.549,-71.911,-178.432,9.988,149.561
C02745=1117.412,255.301,-71.882,-178.433,9.986,149.561
C02746=1117.417,255.053,-71.854,-178.434,9.984,149.560
C02747=1117.422,254.804,-71.825,-178.436,9.982,149.560
C02748=1117.425,254.556,-71.796,-178.437,9.981,149.560
C02749=1117.430,254.308,-71.768,-178.439,9.979,149.561
C02750=1117.434,254.094,-71.742,-178.441,9.977,149.560
C02751=1117.437,253.882,-71.718,-178.443,9.975,149.561
C02752=1117.441,253.668,-71.694,-178.444,9.974,149.561
C02753=1117.445,253.456,-71.670,-178.446,9.972,149.561
C02754=1117.448,253.242,-71.644,-178.448,9.969,149.561
C02755=1117.453,253.029,-71.620,-178.450,9.968,149.561
C02756=1117.455,252.816,-71.596,-178.452,9.966,149.561
C02757=1117.460,252.603,-71.571,-178.455,9.964,149.561
C02758=1117.463,252.354,-71.543,-178.458,9.961,149.561
C02759=1117.468,252.106,-71.514,-178.461,9.959,149.561
C02760=1117.472,251.858,-71.485,-178.463,9.957,149.562
C02761=1117.476,251.609,-71.457,-178.466,9.954,149.562
C02762=1117.480,251.361,-71.429,-178.470,9.952,149.562
C02763=1117.485,251.113,-71.400,-178.473,9.948,149.562
C02764=1117.489,250.864,-71.372,-178.477,9.946,149.562
C02765=1117.494,250.616,-71.343,-178.480,9.943,149.563
C02766=1117.497,250.368,-71.315,-178.483,9.940,149.563
C02767=1117.502,250.119,-71.286,-178.487,9.937,149.563
C02768=1117.506,249.871,-71.258,-178.491,9.934,149.563
C02769=1117.511,249.622,-71.230,-178.495,9.930,149.564
C02770=1117.515,249.374,-71.202,-178.499,9.927,149.564
C02771=1117.520,249.125,-71.173,-178.504,9.923,149.564
C02772=1117.523,248.877,-71.145,-178.508,9.920,149.564
C02773=1117.528,248.629,-71.117,-178.512,9.916,149.565
C02774=1117.532,248.380,-71.088,-178.517,9.912,149.565
C02775=1117.537,248.132,-71.061,-178.521,9.908,149.565
C02776=1117.541,247.883,-71.032,-178.526,9.904,149.565
C02777=1117.545,247.635,-71.004,-178.531,9.900,149.566
C02778=1117.549,247.387,-70.976,-178.534,9.897,149.566
C02779=1117.554,247.139,-70.948,-178.536,9.894,149.566
C02780=1117.558,246.890,-70.919,-178.538,9.892,149.566
C02781=1117.562,246.642,-70.892,-178.540,9.890,149.566
C02782=1117.566,246.394,-70.864,-178.543,9.886,149.566
C02783=1117.571,246.146,-70.835,-178.544,9.884,149.565
C02784=1117.575,245.897,-70.807,-178.546,9.882,149.565
C02785=1117.579,245.649,-70.779,-178.548,9.879,149.565
C02786=1117.584,245.400,-70.751,-178.550,9.877,149.565
C02787=1117.588,245.152,-70.723,-178.553,9.874,149.565
C02788=1117.592,244.903,-70.695,-178.555,9.872,149.565
C02789=1117.596,244.655,-70.668,-178.556,9.869,149.565
C02790=1117.602,244.407,-70.639,-178.558,9.867,149.565
C02791=1117.605,244.158,-70.611,-178.561,9.864,149.565
C02792=1117.610,243.910,-70.584,-178.563,9.862,149.565
C02793=1117.614,243.661,-70.556,-178.565,9.860,149.565
C02794=1117.619,243.413,-70.527,-178.567,9.857,149.565
C02795=1117.623,243.165,-70.499,-178.569,9.854,149.565
C02796=1117.627,242.916,-70.472,-178.572,9.852,149.565
C02797=1117.631,242.668,-70.444,-178.574,9.850,149.565
C02798=1117.635,242.420,-70.416,-178.577,9.847,149.565
C02799=1117.641,242.171,-70.389,-178.578,9.845,149.565
C02800=1117.644,241.922,-70.361,-178.581,9.842,149.565
C02801=1117.649,241.674,-70.333,-178.583,9.840,149.565
C02802=1117.653,241.426,-70.305,-178.585,9.837,149.565
C02803=1117.657,241.177,-70.278,-178.588,9.835,149.565
C02804=1117.661,240.929,-70.249,-178.590,9.832,149.565
C02805=1117.666,240.680,-70.222,-178.593,9.829,149.565
C02806=1117.670,240.468,-70.198,-178.595,9.827,149.565
C02807=1117.674,240.255,-70.174,-178.597,9.825,149.565
C02808=1117.677,240.041,-70.150,-178.600,9.823,149.565
C02809=1117.680,239.828,-70.127,-178.601,9.821,149.565
C02810=1117.685,239.614,-70.103,-178.604,9.819,149.566
C02811=1117.688,239.401,-70.079,-178.606,9.817,149.565
C02812=1117.692,239.188,-70.055,-178.608,9.815,149.566
C02813=1117.695,238.975,-70.032,-178.610,9.813,149.566
C02814=1117.700,238.726,-70.005,-178.613,9.809,149.566
C02815=1117.704,238.478,-69.976,-178.615,9.807,149.566
C02816=1117.709,238.229,-69.949,-178.618,9.805,149.566
C02817=1117.712,237.981,-69.921,-178.621,9.802,149.566
C02818=1117.717,237.732,-69.894,-178.623,9.800,149.566
C02819=1117.721,237.484,-69.866,-178.626,9.797,149.566
C02820=1117.727,237.235,-69.839,-178.629,9.794,149.566
C02821=1117.730,236.987,-69.811,-178.631,9.792,149.566
C02822=1117.735,236.738,-69.784,-178.634,9.789,149.566
C02823=1117.739,236.490,-69.756,-178.637,9.786,149.566
C02824=1117.743,236.241,-69.728,-178.640,9.784,149.567
C02825=1117.748,235.993,-69.701,-178.642,9.782,149.567
C02826=1117.752,235.745,-69.673,-178.645,9.779,149.567
C02827=1117.756,235.496,-69.647,-178.648,9.776,149.567
C02828=1117.760,235.248,-69.619,-178.651,9.773,149.567
C02829=1117.765,235.000,-69.592,-178.653,9.770,149.567
C02830=1117.769,234.751,-69.565,-178.656,9.768,149.567
C02831=1117.773,234.503,-69.537,-178.659,9.765,149.567
C02832=1117.778,234.254,-69.510,-178.662,9.762,149.567
C02833=1117.783,234.006,-69.482,-178.665,9.759,149.568
C02834=1117.786,233.757,-69.454,-178.668,9.757,149.568
C02835=1117.791,233.508,-69.427,-178.671,9.754,149.568
C02836=1117.796,233.260,-69.400,-178.674,9.751,149.568
C02837=1117.800,233.011,-69.373,-178.676,9.748,149.568
C02838=1117.804,232.764,-69.346,-178.679,9.745,149.568
C02839=1117.808,232.515,-69.319,-178.682,9.742,149.568
C02840=1117.813,232.266,-69.291,-178.685,9.740,149.568
C02841=1117.817,232.018,-69.264,-178.688,9.737,149.568
C02842=1117.822,231.769,-69.237,-178.691,9.734,149.568
C02843=1117.826,231.520,-69.210,-178.695,9.731,149.569
C02844=1117.830,231.272,-69.183,-178.698,9.728,149.569
C02845=1117.834,231.024,-69.156,-178.700,9.725,149.569
C02846=1117.839,230.775,-69.129,-178.703,9.722,149.569
C02847=1117.844,230.527,-69.102,-178.707,9.719,149.569
C02848=1117.848,230.278,-69.075,-178.710,9.716,149.569
C02849=1117.852,230.030,-69.048,-178.713,9.713,149.569
C02850=1117.856,229.781,-69.021,-178.716,9.709,149.569
C02851=1117.861,229.533,-68.994,-178.719,9.707,149.569
C02852=1117.865,229.284,-68.967,-178.722,9.703,149.569
C02853=1117.869,229.036,-68.940,-178.725,9.700,149.569
C02854=1117.874,228.787,-68.913,-178.728,9.697,149.570
C02855=1117.879,228.539,-68.886,-178.731,9.693,149.569
C02856=1117.883,228.290,-68.858,-178.734,9.691,149.570
C02857=1117.887,228.042,-68.832,-178.738,9.687,149.570
C02858=1117.891,227.793,-68.805,-178.740,9.684,149.570
C02859=1117.896,227.545,-68.778,-178.743,9.681,149.570
C02860=1117.900,227.296,-68.751,-178.746,9.678,149.570
C02861=1117.905,227.048,-68.724,-178.749,9.675,149.570
C02862=1117.909,226.834,-68.702,-178.751,9.672,149.570
C02863=1117.912,226.621,-68.678,-178.754,9.669,149.570
C02864=1117.916,226.408,-68.656,-178.757,9.667,149.570
C02865=1117.920,226.194,-68.633,-178.759,9.664,149.570
C02866=1117.923,225.981,-68.610,-178.761,9.661,149.570
C02867=1117.927,225.768,-68.587,-178.764,9.658,149.570
C02868=1117.932,225.554,-68.564,-178.766,9.656,149.570
C02869=1117.934,225.341,-68.541,-178.769,9.653,149.570
C02870=1117.939,225.092,-68.515,-178.772,9.650,149.570
C02871=1117.944,224.844,-68.488,-178.774,9.647,149.570
C02872=1117.947,224.595,-68.461,-178.777,9.643,149.570
C02873=1117.952,224.346,-68.434,-178.780,9.640,149.570
C02874=1117.956,224.097,-68.408,-178.782,9.637,149.570
C02875=1117.961,223.849,-68.381,-178.785,9.634,149.569
C02876=1117.965,223.601,-68.355,-178.788,9.631,149.570
C02877=1117.970,223.352,-68.327,-178.790,9.628,149.570
C02878=1117.974,223.103,-68.302,-178.793,9.625,149.569
C02879=1117.978,222.855,-68.275,-178.795,9.622,149.569
C02880=1117.983,222.606,-68.249,-178.798,9.618,149.569
C02881=1117.987,222.358,-68.222,-178.801,9.615,149.569
C02882=1117.991,222.109,-68.195,-178.804,9.612,149.569
C02883=1117.996,221.860,-68.169,-178.806,9.609,149.569
C02884=1118.000,221.612,-68.143,-178.809,9.605,149.569
C02885=1118.006,221.364,-68.117,-178.811,9.602,149.569
C02886=1118.010,221.116,-68.090,-178.814,9.599,149.569
C02887=1118.014,220.867,-68.064,-178.816,9.596,149.569
C02888=1118.018,220.618,-68.037,-178.819,9.593,149.569
C02889=1118.022,220.370,-68.011,-178.821,9.590,149.569
C02890=1118.027,220.121,-67.984,-178.823,9.587,149.568
C02891=1118.031,219.873,-67.958,-178.825,9.584,149.568
C02892=1118.036,219.624,-67.932,-178.828,9.581,149.568
C02893=1118.040,219.375,-67.905,-178.830,9.578,149.568
C02894=1118.044,219.127,-67.879,-178.833,9.575,149.568
C02895=1118.049,218.878,-67.852,-178.835,9.571,149.568
C02896=1118.053,218.629,-67.827,-178.837,9.568,149.568
C02897=1118.057,218.381,-67.801,-178.839,9.566,149.568
C02898=1118.062,218.132,-67.774,-178.842,9.563,149.568
C02899=1118.067,217.884,-67.748,-178.844,9.560,149.568
C02900=1118.071,217.636,-67.722,-178.846,9.556,149.567
C02901=1118.076,217.387,-67.696,-178.849,9.553,149.567
C02902=1118.080,217.138,-67.670,-178.851,9.551,149.567
C02903=1118.084,216.890,-67.643,-178.853,9.547,149.567
C02904=1118.088,216.641,-67.618,-178.855,9.544,149.567
C02905=1118.093,216.392,-67.591,-178.857,9.542,149.567
C02906=1118.097,216.144,-67.565,-178.860,9.539,149.567
C02907=1118.102,215.895,-67.539,-178.862,9.535,149.567
C02908=1118.106,215.647,-67.514,-178.864,9.533,149.567
C02909=1118.111,215.398,-67.487,-178.866,9.530,149.567
C02910=1118.115,215.149,-67.461,-178.868,9.527,149.566
C02911=1118.119,214.901,-67.435,-178.870,9.524,149.566
C02912=1118.123,214.652,-67.409,-178.872,9.522,149.566
C02913=1118.129,214.404,-67.383,-178.874,9.518,149.566
C02914=1118.133,214.155,-67.357,-178.876,9.516,149.566
C02915=1118.137,213.906,-67.331,-178.879,9.513,149.566
C02916=1118.141,213.658,-67.305,-178.880,9.510,149.566
C02917=1118.146,213.409,-67.280,-178.883,9.507,149.566
C02918=1118.150,213.195,-67.257,-178.885,9.505,149.565
C02919=1118.154,212.982,-67.235,-178.887,9.502,149.565
C02920=1118.158,212.769,-67.212,-178.889,9.499,149.565
C02921=1118.161,212.555,-67.191,-178.891,9.497,149.565
C02922=1118.165,212.341,-67.168,-178.893,9.494,149.565
C02923=1118.169,212.128,-67.146,-178.895,9.492,149.565
C02924=1118.173,211.914,-67.123,-178.897,9.489,149.565
C02925=1118.177,211.701,-67.102,-178.899,9.487,149.565
C02926=1118.181,211.452,-67.076,-178.902,9.484,149.565
C02927=1118.185,211.204,-67.050,-178.905,9.481,149.565
C02928=1118.189,210.955,-67.024,-178.907,9.478,149.565
C02929=1118.194,210.707,-66.999,-178.909,9.475,149.565
C02930=1118.199,210.458,-66.972,-178.912,9.473,149.565
C02931=1118.203,210.209,-66.946,-178.915,9.470,149.565
C02932=1118.207,209.960,-66.921,-178.917,9.466,149.565
C02933=1118.212,209.712,-66.895,-178.920,9.464,149.565
C02934=1118.216,209.463,-66.870,-178.923,9.461,149.565
C02935=1118.221,209.215,-66.844,-178.926,9.458,149.565
C02936=1118.225,208.966,-66.818,-178.928,9.455,149.565
C02937=1118.230,208.718,-66.793,-178.930,9.453,149.565
C02938=1118.234,208.469,-66.767,-178.933,9.450,149.565
C02939=1118.238,208.220,-66.741,-178.936,9.447,149.566
C02940=1118.243,207.971,-66.717,-178.938,9.444,149.565
C02941=1118.248,207.723,-66.691,-178.941,9.441,149.566
C02942=1118.252,207.474,-66.665,-178.944,9.438,149.566
C02943=1118.257,207.226,-66.640,-178.947,9.435,149.566
C02944=1118.261,206.977,-66.614,-178.950,9.432,149.566
C02945=1118.265,206.728,-66.588,-178.953,9.430,149.566
C02946=1118.270,206.480,-66.563,-178.955,9.427,149.566
C02947=1118.274,206.231,-66.538,-178.958,9.424,149.566
C02948=1118.279,205.982,-66.512,-178.961,9.421,149.566
C02949=1118.283,205.734,-66.487,-178.964,9.418,149.566
C02950=1118.288,205.485,-66.461,-178.967,9.415,149.566
C02951=1118.293,205.237,-66.435,-178.970,9.413,149.566
C02952=1118.297,204.987,-66.410,-178.973,9.410,149.567
C02953=1118.301,204.738,-66.385,-178.975,9.407,149.567
C02954=1118.305,204.491,-66.360,-178.978,9.404,149.567
C02955=1118.310,204.241,-66.335,-178.981,9.401,149.567
C02956=1118.314,203.992,-66.309,-178.984,9.398,149.567
C02957=1118.319,203.744,-66.284,-178.987,9.395,149.567
C02958=1118.323,203.495,-66.259,-178.990,9.392,149.567
C02959=1118.328,203.247,-66.233,-178.993,9.389,149.567
C02960=1118.333,202.998,-66.208,-178.996,9.386,149.567
C02961=1118.337,202.750,-66.183,-178.998,9.383,149.567
C02962=1118.341,202.501,-66.158,-179.001,9.380,149.567
C02963=1118.345,202.252,-66.132,-179.005,9.377,149.568
C02964=1118.351,202.003,-66.107,-179.008,9.374,149.568
C02965=1118.355,201.754,-66.082,-179.011,9.371,149.568
C02966=1118.359,201.506,-66.057,-179.013,9.368,149.568
C02967=1118.363,201.257,-66.032,-179.017,9.365,149.568
C02968=1118.368,201.009,-66.007,-179.020,9.362,149.568
C02969=1118.373,200.760,-65.981,-179.023,9.359,149.568
C02970=1118.377,200.511,-65.957,-179.026,9.355,149.568
C02971=1118.381,200.263,-65.931,-179.029,9.353,149.568
C02972=1118.386,200.014,-65.907,-179.032,9.350,149.568
C02973=1118.390,199.765,-65.882,-179.035,9.346,149.568
C02974=1118.394,199.551,-65.860,-179.037,9.344,149.569
C02975=1118.398,199.338,-65.838,-179.040,9.341,149.569
C02976=1118.402,199.124,-65.817,-179.043,9.338,149.569
C02977=1118.406,198.911,-65.796,-179.046,9.336,149.569
C02978=1118.410,198.697,-65.774,-179.048,9.332,149.569
C02979=1118.414,198.483,-65.753,-179.051,9.330,149.569
C02980=1118.418,198.269,-65.732,-179.053,9.327,149.569
C02981=1118.421,198.055,-65.710,-179.056,9.325,149.569
C02982=1118.425,197.808,-65.686,-179.059,9.321,149.569
C02983=1118.430,197.558,-65.660,-179.062,9.318,149.569
C02984=1118.435,197.310,-65.636,-179.065,9.314,149.569
C02985=1118.439,197.062,-65.611,-179.069,9.311,149.569
C02986=1118.444,196.812,-65.586,-179.072,9.308,149.569
C02987=1118.448,196.564,-65.562,-179.075,9.304,149.569
C02988=1118.453,196.314,-65.537,-179.078,9.301,149.569
C02989=1118.457,196.067,-65.512,-179.080,9.298,149.569
C02990=1118.461,195.817,-65.487,-179.082,9.295,149.569
C02991=1118.466,195.569,-65.462,-179.084,9.293,149.569
C02992=1118.471,195.320,-65.438,-179.085,9.290,149.569
C02993=1118.475,195.071,-65.413,-179.088,9.287,149.569
C02994=1118.479,194.823,-65.388,-179.089,9.284,149.568
C02995=1118.485,194.574,-65.364,-179.091,9.282,149.568
C02996=1118.488,194.325,-65.339,-179.093,9.279,149.568
C02997=1118.493,194.076,-65.315,-179.095,9.276,149.568
C02998=1118.497,193.827,-65.290,-179.097,9.274,149.568
C02999=1118.502,193.578,-65.266,-179.099,9.271,149.568
C03000=1118.507,193.330,-65.242,-179.101,9.268,149.568
C03001=1118.511,193.081,-65.216,-179.103,9.266,149.568
C03002=1118.515,192.833,-65.192,-179.105,9.263,149.568
C03003=1118.521,192.584,-65.167,-179.107,9.260,149.568
C03004=1118.524,192.335,-65.143,-179.109,9.258,149.568
C03005=1118.529,192.086,-65.118,-179.111,9.254,149.567
C03006=1118.534,191.838,-65.094,-179.113,9.252,149.567
C03007=1118.538,191.589,-65.069,-179.116,9.249,149.567
C03008=1118.543,191.340,-65.045,-179.117,9.247,149.567
C03009=1118.547,191.092,-65.021,-179.120,9.243,149.567
C03010=1118.552,190.842,-64.996,-179.122,9.241,149.567
C03011=1118.556,190.594,-64.972,-179.124,9.239,149.567
C03012=1118.561,190.345,-64.947,-179.126,9.235,149.567
C03013=1118.565,190.096,-64.922,-179.128,9.233,149.567
C03014=1118.569,189.848,-64.898,-179.130,9.230,149.567
C03015=1118.575,189.599,-64.874,-179.133,9.227,149.567
C03016=1118.579,189.350,-64.850,-179.135,9.224,149.567
C03017=1118.583,189.101,-64.825,-179.137,9.221,149.567
C03018=1118.588,188.852,-64.801,-179.139,9.219,149.567
C03019=1118.593,188.604,-64.777,-179.142,9.216,149.566
C03020=1118.598,188.355,-64.752,-179.143,9.214,149.566
C03021=1118.601,188.106,-64.728,-179.146,9.210,149.566
C03022=1118.606,187.857,-64.704,-179.149,9.207,149.566
C03023=1118.611,187.609,-64.679,-179.150,9.205,149.566
C03024=1118.615,187.360,-64.655,-179.153,9.202,149.566
C03025=1118.619,187.110,-64.632,-179.155,9.199,149.566
C03026=1118.625,186.862,-64.607,-179.157,9.196,149.566
C03027=1118.629,186.613,-64.583,-179.160,9.194,149.566
C03028=1118.633,186.365,-64.559,-179.163,9.191,149.566
C03029=1118.637,186.116,-64.534,-179.165,9.188,149.566
C03030=1118.642,185.902,-64.514,-179.167,9.185,149.566
C03031=1118.646,185.689,-64.493,-179.169,9.183,149.566
C03032=1118.649,185.474,-64.473,-179.171,9.181,149.566
C03033=1118.653,185.261,-64.451,-179.174,9.177,149.566
C03034=1118.657,185.047,-64.431,-179.175,9.175,149.566
C03035=1118.661,184.834,-64.410,-179.177,9.173,149.566
C03036=1118.665,184.620,-64.390,-179.179,9.170,149.566
C03037=1118.669,184.406,-64.368,-179.182,9.167,149.566
C03038=1118.674,184.157,-64.345,-179.185,9.165,149.566
C03039=1118.678,183.908,-64.321,-179.187,9.161,149.566
C03040=1118.682,183.660,-64.297,-179.189,9.159,149.566
C03041=1118.688,183.411,-64.273,-179.192,9.156,149.566
C03042=1118.692,183.161,-64.248,-179.194,9.153,149.566
C03043=1118.696,182.913,-64.224,-179.197,9.150,149.566
C03044=1118.701,182.664,-64.201,-179.199,9.147,149.566
C03045=1118.705,182.416,-64.177,-179.202,9.144,149.566
C03046=1118.710,182.167,-64.154,-179.204,9.140,149.566
C03047=1118.714,181.918,-64.129,-179.207,9.138,149.566
C03048=1118.720,181.669,-64.106,-179.210,9.135,149.566
C03049=1118.724,181.420,-64.081,-179.212,9.132,149.566
C03050=1118.728,181.171,-64.058,-179.215,9.128,149.566
C03051=1118.732,180.922,-64.034,-179.218,9.125,149.566
C03052=1118.737,180.673,-64.010,-179.220,9.121,149.566
C03053=1118.742,180.425,-63.986,-179.223,9.118,149.566
C03054=1118.746,180.176,-63.963,-179.226,9.115,149.566
C03055=1118.751,179.927,-63.939,-179.228,9.112,149.566
C03056=1118.755,179.678,-63.915,-179.231,9.108,149.566
C03057=1118.760,179.430,-63.891,-179.234,9.105,149.565
C03058=1118.764,179.181,-63.868,-179.236,9.102,149.565
C03059=1118.769,178.932,-63.844,-179.238,9.100,149.565
C03060=1118.773,178.683,-63.820,-179.241,9.097,149.565
C03061=1118.778,178.434,-63.797,-179.243,9.093,149.565
C03062=1118.782,178.185,-63.773,-179.245,9.091,149.565
C03063=1118.787,177.936,-63.749,-179.247,9.088,149.565
C03064=1118.791,177.687,-63.726,-179.249,9.084,149.565
C03065=1118.796,177.439,-63.702,-179.251,9.082,149.565
C03066=1118.801,177.190,-63.679,-179.254,9.079,149.565
C03067=1118.805,176.941,-63.655,-179.255,9.076,149.564
C03068=1118.810,176.692,-63.631,-179.258,9.073,149.564
C03069=1118.814,176.443,-63.608,-179.260,9.070,149.564
C03070=1118.819,176.194,-63.584,-179.262,9.067,149.564
C03071=1118.823,175.946,-63.560,-179.264,9.064,149.564
C03072=1118.828,175.697,-63.537,-179.267,9.061,149.564
C03073=1118.833,175.448,-63.514,-179.268,9.058,149.564
C03074=1118.837,175.199,-63.491,-179.271,9.055,149.564
C03075=1118.841,174.950,-63.468,-179.273,9.052,149.564
C03076=1118.846,174.702,-63.443,-179.275,9.049,149.564
C03077=1118.851,174.453,-63.420,-179.277,9.046,149.564
C03078=1118.855,174.204,-63.397,-179.280,9.043,149.563
C03079=1118.860,173.955,-63.373,-179.282,9.041,149.563
C03080=1118.865,173.706,-63.350,-179.284,9.037,149.563
C03081=1118.869,173.457,-63.326,-179.286,9.034,149.563
C03082=1118.873,173.208,-63.303,-179.289,9.031,149.563
C03083=1118.878,172.959,-63.280,-179.290,9.028,149.563
C03084=1118.883,172.711,-63.257,-179.293,9.025,149.563
C03085=1118.888,172.462,-63.233,-179.295,9.022,149.563
C03086=1118.893,172.136,-63.203,-179.298,9.018,149.563
C03087=1118.900,171.810,-63.172,-179.300,9.015,149.563
C03088=1118.905,171.485,-63.142,-179.304,9.011,149.562
C03089=1118.911,171.159,-63.112,-179.306,9.007,149.562
C03090=1118.916,170.910,-63.089,-179.309,9.003,149.562
C03091=1118.921,170.661,-63.065,-179.311,9.000,149.562
C03092=1118.925,170.412,-63.042,-179.313,8.998,149.562
C03093=1118.930,170.164,-63.020,-179.315,8.995,149.562
C03094=1118.934,169.915,-62.996,-179.318,8.991,149.562
C03095=1118.939,169.666,-62.973,-179.320,8.988,149.562
C03096=1118.944,169.417,-62.949,-179.322,8.986,149.562
C03097=1118.948,169.168,-62.927,-179.324,8.983,149.562
C03098=1118.953,168.919,-62.903,-179.327,8.979,149.561
C03099=1118.957,168.670,-62.880,-179.329,8.976,149.561
C03100=1118.962,168.422,-62.858,-179.332,8.973,149.561
C03101=1118.967,168.173,-62.834,-179.333,8.970,149.561
C03102=1118.971,167.924,-62.811,-179.336,8.967,149.561
C03103=1118.975,167.674,-62.789,-179.338,8.964,149.561
C03104=1118.980,167.425,-62.765,-179.341,8.961,149.561
C03105=1118.985,167.176,-62.742,-179.343,8.957,149.561
C03106=1118.992,166.826,-62.710,-179.346,8.953,149.561
C03107=1118.998,166.475,-62.678,-179.349,8.949,149.560
C03108=1119.004,166.124,-62.645,-179.352,8.944,149.560
C03109=1119.010,165.773,-62.613,-179.355,8.940,149.560
C03110=1119.016,165.525,-62.590,-179.358,8.937,149.560
C03111=1119.020,165.275,-62.568,-179.360,8.934,149.560
C03112=1119.025,165.026,-62.544,-179.362,8.931,149.560
C03113=1119.029,164.777,-62.522,-179.365,8.927,149.560
C03114=1119.033,164.528,-62.498,-179.367,8.925,149.560
C03115=1119.038,164.280,-62.477,-179.369,8.922,149.559
C03116=1119.043,164.031,-62.453,-179.371,8.918,149.559
C03117=1119.048,163.782,-62.430,-179.374,8.915,149.559
C03118=1119.052,163.532,-62.408,-179.376,8.912,149.559
C03119=1119.057,163.284,-62.385,-179.378,8.909,149.559
C03120=1119.061,163.035,-62.362,-179.380,8.905,149.559
C03121=1119.066,162.786,-62.339,-179.383,8.902,149.559
C03122=1119.070,162.537,-62.317,-179.385,8.899,149.559
C03123=1119.076,162.288,-62.294,-179.388,8.896,149.559
C03124=1119.080,162.039,-62.272,-179.389,8.893,149.558
C03125=1119.084,161.791,-62.249,-179.392,8.890,149.558
C03126=1119.089,161.542,-62.227,-179.394,8.887,149.558
C03127=1119.093,161.293,-62.204,-179.397,8.884,149.558
C03128=1119.098,161.043,-62.181,-179.399,8.880,149.558
C03129=1119.102,160.795,-62.158,-179.401,8.877,149.558
C03130=1119.108,160.546,-62.136,-179.403,8.873,149.558
C03131=1119.112,160.297,-62.113,-179.406,8.870,149.558
C03132=1119.117,160.047,-62.091,-179.408,8.867,149.558
C03133=1119.121,159.799,-62.068,-179.410,8.864,149.557
C03134=1119.126,159.550,-62.046,-179.413,8.861,149.557
C03135=1119.130,159.301,-62.023,-179.415,8.857,149.557
C03136=1119.135,159.052,-62.001,-179.417,8.854,149.557
C03137=1119.139,158.803,-61.978,-179.420,8.851,149.557
C03138=1119.143,158.589,-61.959,-179.422,8.847,149.557
C03139=1119.147,158.375,-61.940,-179.424,8.845,149.557
C03140=1119.151,158.161,-61.921,-179.425,8.842,149.557
C03141=1119.155,157.947,-61.901,-179.428,8.839,149.557
C03142=1119.159,157.733,-61.882,-179.429,8.837,149.556
C03143=1119.163,157.519,-61.863,-179.432,8.834,149.556
C03144=1119.167,157.305,-61.843,-179.433,8.831,149.556
C03145=1119.171,157.091,-61.824,-179.436,8.828,149.556
C03146=1119.176,156.843,-61.803,-179.438,8.824,149.556
C03147=1119.181,156.593,-61.780,-179.441,8.821,149.556
C03148=1119.186,156.345,-61.758,-179.443,8.818,149.555
C03149=1119.190,156.096,-61.736,-179.445,8.814,149.555
C03150=1119.194,155.846,-61.713,-179.447,8.811,149.555
C03151=1119.200,155.598,-61.690,-179.450,8.808,149.555
C03152=1119.204,155.349,-61.668,-179.452,8.804,149.555
C03153=1119.209,155.100,-61.647,-179.454,8.801,149.555
C03154=1119.213,154.851,-61.625,-179.457,8.797,149.555
C03155=1119.219,154.602,-61.602,-179.459,8.794,149.554
C03156=1119.222,154.353,-61.580,-179.462,8.790,149.554
C03157=1119.227,154.104,-61.558,-179.464,8.787,149.554
C03158=1119.232,153.855,-61.536,-179.466,8.783,149.554
C03159=1119.236,153.606,-61.514,-179.468,8.780,149.554
C03160=1119.242,153.357,-61.492,-179.470,8.777,149.554
C03161=1119.246,153.107,-61.470,-179.473,8.773,149.553
C03162=1119.250,152.859,-61.447,-179.476,8.769,149.553
C03163=1119.255,152.610,-61.425,-179.478,8.766,149.553
C03164=1119.259,152.361,-61.403,-179.480,8.763,149.553
C03165=1119.264,152.112,-61.381,-179.482,8.759,149.553
C03166=1119.269,151.863,-61.359,-179.485,8.755,149.553
C03167=1119.274,151.614,-61.337,-179.487,8.752,149.552
C03168=1119.278,151.365,-61.315,-179.489,8.748,149.552
C03169=1119.283,151.116,-61.293,-179.492,8.745,149.552
C03170=1119.288,150.867,-61.272,-179.494,8.741,149.552
C03171=1119.292,150.618,-61.250,-179.497,8.737,149.552
C03172=1119.297,150.369,-61.228,-179.499,8.734,149.551
C03173=1119.302,150.120,-61.206,-179.501,8.731,149.551
C03174=1119.306,149.871,-61.184,-179.504,8.726,149.551
C03175=1119.311,149.622,-61.163,-179.506,8.723,149.551
C03176=1119.316,149.373,-61.140,-179.508,8.719,149.551
C03177=1119.321,149.124,-61.118,-179.510,8.716,149.550
C03178=1119.325,148.875,-61.096,-179.513,8.712,149.550
C03179=1119.330,148.626,-61.074,-179.515,8.709,149.550
C03180=1119.335,148.377,-61.053,-179.517,8.705,149.550
C03181=1119.339,148.128,-61.031,-179.520,8.701,149.550
C03182=1119.344,147.879,-61.010,-179.522,8.697,149.550
C03183=1119.348,147.630,-60.988,-179.524,8.694,149.549
C03184=1119.353,147.381,-60.966,-179.527,8.690,149.549
C03185=1119.358,147.132,-60.944,-179.529,8.686,149.549
C03186=1119.362,146.883,-60.924,-179.531,8.683,149.549
C03187=1119.367,146.634,-60.902,-179.534,8.678,149.548
C03188=1119.371,146.385,-60.880,-179.536,8.675,149.548
C03189=1119.376,146.136,-60.858,-179.539,8.671,149.548
C03190=1119.381,145.887,-60.837,-179.541,8.668,149.548
C03191=1119.385,145.637,-60.815,-179.543,8.664,149.548
C03192=1119.390,145.389,-60.793,-179.546,8.659,149.547
C03193=1119.395,145.140,-60.772,-179.548,8.656,149.547
C03194=1119.400,144.925,-60.753,-179.549,8.653,149.547
C03195=1119.403,144.711,-60.735,-179.550,8.650,149.546
C03196=1119.408,144.498,-60.716,-179.552,8.647,149.546
C03197=1119.411,144.283,-60.698,-179.554,8.644,149.546
C03198=1119.415,144.069,-60.679,-179.555,8.641,149.546
C03199=1119.419,143.855,-60.661,-179.556,8.638,149.545
C03200=1119.424,143.641,-60.643,-179.557,8.635,149.545
C03201=1119.427,143.427,-60.624,-179.559,8.633,149.545
C03202=1119.432,143.178,-60.603,-179.560,8.630,149.544
C03203=1119.436,142.929,-60.581,-179.562,8.626,149.544
C03204=1119.441,142.680,-60.560,-179.564,8.622,149.544
C03205=1119.446,142.431,-60.539,-179.565,8.619,149.543
C03206=1119.450,142.182,-60.517,-179.567,8.616,149.543
C03207=1119.455,141.933,-60.496,-179.568,8.613,149.543
C03208=1119.460,141.684,-60.475,-179.570,8.609,149.542
C03209=1119.465,141.435,-60.454,-179.571,8.605,149.542
C03210=1119.469,141.186,-60.432,-179.573,8.602,149.542
C03211=1119.474,140.937,-60.411,-179.575,8.599,149.541
C03212=1119.479,140.688,-60.390,-179.576,8.596,149.541
C03213=1119.484,140.439,-60.368,-179.578,8.592,149.541
C03214=1119.487,140.190,-60.347,-179.579,8.589,149.540
C03215=1119.492,139.941,-60.325,-179.581,8.586,149.540
C03216=1119.498,139.692,-60.304,-179.583,8.582,149.540
C03217=1119.502,139.443,-60.283,-179.584,8.579,149.539
C03218=1119.506,139.193,-60.262,-179.586,8.575,149.539
C03219=1119.511,138.944,-60.241,-179.587,8.573,149.539
C03220=1119.516,138.695,-60.219,-179.589,8.569,149.538
C03221=1119.521,138.447,-60.199,-179.591,8.565,149.538
C03222=1119.525,138.197,-60.177,-179.592,8.563,149.538
C03223=1119.530,137.948,-60.156,-179.594,8.559,149.537
C03224=1119.535,137.699,-60.135,-179.596,8.556,149.537
C03225=1119.539,137.450,-60.114,-179.597,8.552,149.537
C03226=1119.545,137.201,-60.093,-179.599,8.549,149.536
C03227=1119.548,136.952,-60.072,-179.601,8.546,149.536
C03228=1119.553,136.703,-60.051,-179.602,8.542,149.536
C03229=1119.559,136.454,-60.030,-179.604,8.539,149.536
C03230=1119.563,136.205,-60.009,-179.605,8.535,149.535
C03231=1119.568,135.956,-59.988,-179.608,8.532,149.535
C03232=1119.573,135.707,-59.967,-179.609,8.529,149.535
C03233=1119.577,135.457,-59.946,-179.611,8.525,149.534
C03234=1119.582,135.208,-59.924,-179.612,8.523,149.534
C03235=1119.586,134.959,-59.904,-179.614,8.519,149.534
C03236=1119.591,134.710,-59.883,-179.616,8.515,149.533
C03237=1119.596,134.462,-59.861,-179.617,8.513,149.533
C03238=1119.601,134.213,-59.841,-179.619,8.509,149.533
C03239=1119.606,133.963,-59.820,-179.621,8.505,149.532
C03240=1119.610,133.714,-59.799,-179.622,8.503,149.532
C03241=1119.615,133.464,-59.778,-179.624,8.499,149.532
C03242=1119.619,133.216,-59.757,-179.625,8.496,149.532
C03243=1119.624,132.967,-59.736,-179.627,8.492,149.531
C03244=1119.629,132.718,-59.715,-179.630,8.489,149.531
C03245=1119.634,132.469,-59.695,-179.631,8.486,149.531
C03246=1119.639,132.219,-59.674,-179.633,8.482,149.530
C03247=1119.643,131.970,-59.653,-179.635,8.479,149.530
C03248=1119.648,131.722,-59.632,-179.636,8.476,149.530
C03249=1119.652,131.472,-59.611,-179.638,8.472,149.530
C03250=1119.656,131.258,-59.594,-179.639,8.470,149.529
C03251=1119.661,131.044,-59.575,-179.641,8.467,149.529
C03252=1119.665,130.830,-59.558,-179.642,8.464,149.529
C03253=1119.669,130.615,-59.540,-179.644,8.461,149.529
C03254=1119.673,130.401,-59.523,-179.645,8.459,149.528
C03255=1119.677,130.187,-59.504,-179.647,8.455,149.528
C03256=1119.681,129.973,-59.486,-179.649,8.453,149.528
C03257=1119.685,129.759,-59.468,-179.650,8.449,149.528
C03258=1119.689,129.510,-59.448,-179.652,8.446,149.527
C03259=1119.694,129.261,-59.427,-179.653,8.443,149.527
C03260=1119.699,129.012,-59.407,-179.655,8.440,149.527
C03261=1119.704,128.763,-59.386,-179.657,8.436,149.526
C03262=1119.708,128.514,-59.365,-179.658,8.433,149.526
C03263=1119.714,128.264,-59.344,-179.660,8.430,149.526
C03264=1119.718,128.015,-59.324,-179.662,8.426,149.526
C03265=1119.723,127.766,-59.304,-179.663,8.423,149.525
C03266=1119.728,127.517,-59.283,-179.665,8.420,149.525
C03267=1119.732,127.268,-59.263,-179.667,8.416,149.525
C03268=1119.737,127.019,-59.243,-179.669,8.413,149.525
C03269=1119.742,126.769,-59.222,-179.671,8.409,149.524
C03270=1119.746,126.520,-59.201,-179.673,8.406,149.524
C03271=1119.751,126.272,-59.181,-179.674,8.403,149.524
C03272=1119.756,126.022,-59.160,-179.676,8.400,149.524
C03273=1119.761,125.773,-59.139,-179.678,8.396,149.523
C03274=1119.765,125.524,-59.119,-179.679,8.393,149.523
C03275=1119.770,125.275,-59.098,-179.681,8.390,149.523
C03276=1119.775,125.026,-59.078,-179.683,8.386,149.522
C03277=1119.779,124.777,-59.058,-179.685,8.383,149.522
C03278=1119.785,124.527,-59.037,-179.686,8.380,149.522
C03279=1119.789,124.278,-59.017,-179.688,8.376,149.522
C03280=1119.793,124.029,-58.996,-179.690,8.373,149.521
C03281=1119.798,123.780,-58.977,-179.692,8.370,149.521
C03282=1119.803,123.531,-58.956,-179.694,8.366,149.521
C03283=1119.808,123.282,-58.935,-179.696,8.362,149.520
C03284=1119.812,123.033,-58.915,-179.697,8.360,149.520
C03285=1119.818,122.784,-58.896,-179.699,8.356,149.520
C03286=1119.823,122.535,-58.875,-179.701,8.353,149.520
C03287=1119.827,122.286,-58.854,-179.703,8.349,149.519
C03288=1119.832,122.037,-58.834,-179.704,8.346,149.519
C03289=1119.836,121.787,-58.814,-179.706,8.343,149.519
C03290=1119.841,121.538,-58.794,-179.708,8.339,149.519
C03291=1119.846,121.289,-58.773,-179.709,8.336,149.518
C03292=1119.851,121.039,-58.753,-179.711,8.333,149.518
C03293=1119.855,120.790,-58.733,-179.714,8.329,149.518
C03294=1119.860,120.541,-58.713,-179.716,8.326,149.518
C03295=1119.865,120.293,-58.693,-179.717,8.323,149.517
C03296=1119.869,120.044,-58.673,-179.719,8.319,149.517
C03297=1119.875,119.794,-58.653,-179.721,8.316,149.517
C03298=1119.879,119.545,-58.632,-179.723,8.312,149.516
C03299=1119.884,119.296,-58.612,-179.724,8.309,149.516
C03300=1119.888,119.046,-58.592,-179.726,8.305,149.516
C03301=1119.893,118.797,-58.572,-179.728,8.302,149.516
C03302=1119.898,118.548,-58.553,-179.730,8.298,149.515
C03303=1119.903,118.300,-58.532,-179.732,8.295,149.515
C03304=1119.907,118.050,-58.513,-179.733,8.292,149.515
C03305=1119.912,117.801,-58.492,-179.735,8.288,149.514
C03306=1119.916,117.587,-58.476,-179.737,8.286,149.514
C03307=1119.920,117.372,-58.458,-179.739,8.282,149.514
C03308=1119.924,117.158,-58.440,-179.740,8.279,149.514
C03309=1119.929,116.944,-58.424,-179.741,8.277,149.514
C03310=1119.932,116.729,-58.406,-179.743,8.274,149.513
C03311=1119.937,116.515,-58.389,-179.745,8.270,149.513
C03312=1119.941,116.301,-58.372,-179.746,8.268,149.513
C03313=1119.945,116.086,-58.355,-179.748,8.265,149.513
C03314=1119.950,115.838,-58.335,-179.749,8.261,149.512
C03315=1119.955,115.588,-58.315,-179.751,8.258,149.512
C03316=1119.959,115.339,-58.295,-179.754,8.254,149.512
C03317=1119.964,115.090,-58.275,-179.755,8.251,149.512
C03318=1119.970,114.841,-58.256,-179.757,8.248,149.511
C03319=1119.974,114.592,-58.235,-179.759,8.244,149.511
C03320=1119.979,114.342,-58.216,-179.761,8.241,149.511
C03321=1119.983,114.093,-58.196,-179.763,8.237,149.510
C03322=1119.989,113.845,-58.176,-179.764,8.233,149.510
C03323=1119.993,113.595,-58.156,-179.766,8.230,149.510
C03324=1119.997,113.346,-58.137,-179.768,8.227,149.510
C03325=1120.002,113.097,-58.117,-179.770,8.223,149.509
C03326=1120.007,112.848,-58.098,-179.772,8.220,149.509
C03327=1120.012,112.598,-58.078,-179.774,8.216,149.509
C03328=1120.017,112.349,-58.058,-179.776,8.213,149.509
C03329=1120.022,112.101,-58.038,-179.778,8.209,149.508
C03330=1120.026,111.851,-58.019,-179.779,8.206,149.508
C03331=1120.031,111.601,-57.999,-179.781,8.202,149.508
C03332=1120.036,111.352,-57.979,-179.783,8.199,149.507
C03333=1120.041,111.104,-57.959,-179.784,8.195,149.507
C03334=1120.046,110.854,-57.940,-179.787,8.192,149.507
C03335=1120.050,110.605,-57.921,-179.789,8.187,149.507
C03336=1120.055,110.356,-57.901,-179.791,8.184,149.506
C03337=1120.060,110.106,-57.882,-179.793,8.180,149.506
C03338=1120.064,109.857,-57.862,-179.796,8.176,149.506
C03339=1120.069,109.608,-57.842,-179.798,8.173,149.506
C03340=1120.074,109.359,-57.822,-179.800,8.169,149.505
C03341=1120.079,109.110,-57.804,-179.803,8.165,149.505
C03342=1120.084,108.861,-57.784,-179.805,8.161,149.505
C03343=1120.088,108.611,-57.764,-179.807,8.158,149.505
C03344=1120.094,108.362,-57.745,-179.810,8.153,149.505
C03345=1120.098,108.113,-57.725,-179.811,8.150,149.504
C03346=1120.102,107.864,-57.706,-179.813,8.146,149.504
C03347=1120.108,107.615,-57.687,-179.816,8.142,149.504
C03348=1120.112,107.365,-57.667,-179.818,8.138,149.503
C03349=1120.118,107.116,-57.648,-179.820,8.135,149.503
C03350=1120.122,106.867,-57.629,-179.822,8.130,149.503
C03351=1120.127,106.617,-57.609,-179.824,8.127,149.503
C03352=1120.132,106.369,-57.590,-179.826,8.123,149.502
C03353=1120.136,106.119,-57.571,-179.828,8.119,149.502
C03354=1120.141,105.870,-57.552,-179.831,8.115,149.502
C03355=1120.146,105.621,-57.532,-179.833,8.111,149.501
C03356=1120.151,105.372,-57.513,-179.834,8.108,149.501
C03357=1120.155,105.123,-57.494,-179.837,8.103,149.501
C03358=1120.161,104.874,-57.475,-179.839,8.100,149.501
C03359=1120.165,104.624,-57.456,-179.841,8.096,149.500
C03360=1120.170,104.374,-57.437,-179.843,8.092,149.500
C03361=1120.175,104.126,-57.417,-179.845,8.088,149.499
C03362=1120.179,103.911,-57.401,-179.846,8.085,149.499
C03363=1120.183,103.697,-57.384,-179.849,8.081,149.499
C03364=1120.187,103.483,-57.368,-179.850,8.078,149.499
C03365=1120.191,103.268,-57.351,-179.852,8.075,149.498
C03366=1120.195,103.054,-57.335,-179.854,8.071,149.498
C03367=1120.200,102.839,-57.318,-179.855,8.069,149.498
C03368=1120.203,102.625,-57.302,-179.857,8.065,149.498
C03369=1120.208,102.411,-57.286,-179.859,8.061,149.497
C03370=1120.212,102.161,-57.267,-179.860,8.057,149.497
C03371=1120.218,101.912,-57.248,-179.862,8.054,149.497
C03372=1120.222,101.663,-57.229,-179.864,8.050,149.496
C03373=1120.227,101.414,-57.210,-179.866,8.046,149.496
C03374=1120.233,101.164,-57.191,-179.868,8.043,149.496
C03375=1120.237,100.915,-57.172,-179.870,8.038,149.495
C03376=1120.242,100.666,-57.153,-179.872,8.034,149.495
C03377=1120.246,100.416,-57.134,-179.874,8.031,149.494
C03378=1120.252,100.168,-57.115,-179.875,8.027,149.494
C03379=1120.256,99.918,-57.096,-179.877,8.023,149.494
C03380=1120.261,99.669,-57.077,-179.879,8.019,149.493
C03381=1120.266,99.420,-57.059,-179.880,8.015,149.493
C03382=1120.271,99.171,-57.039,-179.883,8.011,149.493
C03383=1120.276,98.921,-57.021,-179.885,8.007,149.492
C03384=1120.280,98.672,-57.002,-179.886,8.003,149.492
C03385=1120.285,98.423,-56.984,-179.888,7.999,149.491
C03386=1120.290,98.174,-56.965,-179.889,7.996,149.491
C03387=1120.295,97.924,-56.946,-179.892,7.992,149.491
C03388=1120.299,97.675,-56.927,-179.893,7.988,149.490
C03389=1120.305,97.425,-56.908,-179.895,7.984,149.490
C03390=1120.309,97.177,-56.890,-179.896,7.980,149.490
C03391=1120.314,96.928,-56.872,-179.898,7.976,149.489
C03392=1120.319,96.678,-56.852,-179.900,7.973,149.489
C03393=1120.324,96.429,-56.834,-179.901,7.969,149.488
C03394=1120.328,96.180,-56.815,-179.903,7.964,149.488
C03395=1120.333,95.930,-56.796,-179.905,7.961,149.488
C03396=1120.338,95.681,-56.778,-179.907,7.957,149.487
C03397=1120.343,95.431,-56.759,-179.909,7.953,149.487
C03398=1120.348,95.183,-56.740,-179.910,7.949,149.486
C03399=1120.353,94.934,-56.722,-179.912,7.945,149.486
C03400=1120.358,94.684,-56.703,-179.913,7.941,149.485
C03401=1120.362,94.435,-56.684,-179.915,7.937,149.485
C03402=1120.367,94.186,-56.666,-179.917,7.933,149.485
C03403=1120.372,93.936,-56.648,-179.918,7.929,149.484
C03404=1120.377,93.687,-56.629,-179.920,7.926,149.484
C03405=1120.382,93.438,-56.611,-179.921,7.922,149.483
C03406=1120.387,93.189,-56.593,-179.923,7.918,149.483
C03407=1120.391,92.939,-56.573,-179.924,7.915,149.482
C03408=1120.396,92.690,-56.555,-179.926,7.911,149.482
C03409=1120.401,92.441,-56.537,-179.927,7.906,149.481
C03410=1120.406,92.192,-56.518,-179.928,7.903,149.481
C03411=1120.411,91.942,-56.500,-179.930,7.899,149.480
C03412=1120.416,91.693,-56.482,-179.932,7.895,149.480
C03413=1120.421,91.444,-56.464,-179.933,7.891,149.480
C03414=1120.425,91.195,-56.445,-179.935,7.887,149.479
C03415=1120.430,90.945,-56.426,-179.936,7.883,149.479
C03416=1120.435,90.696,-56.408,-179.938,7.879,149.478
C03417=1120.440,90.446,-56.390,-179.939,7.875,149.478
C03418=1120.444,90.232,-56.374,-179.940,7.872,149.477
C03419=1120.448,90.018,-56.358,-179.941,7.869,149.477
C03420=1120.452,89.803,-56.343,-179.943,7.865,149.477
C03421=1120.457,89.588,-56.326,-179.944,7.862,149.476
C03422=1120.461,89.374,-56.311,-179.945,7.859,149.476
C03423=1120.465,89.160,-56.295,-179.947,7.855,149.475
C03424=1120.469,88.945,-56.280,-179.948,7.852,149.475
C03425=1120.473,88.730,-56.264,-179.948,7.849,149.474
C03426=1120.478,88.481,-56.246,-179.950,7.845,149.474
C03427=1120.482,88.232,-56.227,-179.952,7.841,149.474
C03428=1120.488,87.983,-56.209,-179.953,7.837,149.473
C03429=1120.493,87.734,-56.191,-179.954,7.834,149.473
C03430=1120.498,87.485,-56.173,-179.955,7.830,149.472
C03431=1120.502,87.235,-56.155,-179.957,7.826,149.472
C03432=1120.507,86.986,-56.137,-179.958,7.822,149.471
C03433=1120.512,86.736,-56.119,-179.959,7.819,149.471
C03434=1120.517,86.487,-56.101,-179.961,7.815,149.470
C03435=1120.522,86.238,-56.083,-179.962,7.810,149.469
C03436=1120.527,85.989,-56.065,-179.963,7.806,149.469
C03437=1120.531,85.739,-56.046,-179.964,7.803,149.469
C03438=1120.536,85.490,-56.028,-179.966,7.799,149.468
C03439=1120.541,85.241,-56.010,-179.967,7.795,149.468
C03440=1120.546,84.991,-55.992,-179.969,7.791,149.467
C03441=1120.551,84.742,-55.974,-179.969,7.788,149.466
C03442=1120.556,84.493,-55.956,-179.971,7.784,149.466
C03443=1120.561,84.244,-55.938,-179.972,7.780,149.465
C03444=1120.566,83.994,-55.920,-179.973,7.776,149.465
C03445=1120.571,83.745,-55.902,-179.974,7.773,149.465
C03446=1120.575,83.495,-55.884,-179.976,7.768,149.464
C03447=1120.580,83.246,-55.867,-179.977,7.765,149.463
C03448=1120.585,82.997,-55.849,-179.978,7.761,149.463
C03449=1120.590,82.748,-55.831,-179.979,7.757,149.462
C03450=1120.595,82.498,-55.813,-179.980,7.754,149.462
C03451=1120.600,82.249,-55.795,-179.981,7.750,149.461
C03452=1120.605,82.000,-55.777,-179.982,7.746,149.461
C03453=1120.609,81.751,-55.759,-179.983,7.742,149.460
C03454=1120.615,81.501,-55.742,-179.985,7.738,149.460
C03455=1120.619,81.251,-55.723,-179.986,7.735,149.459
C03456=1120.624,81.002,-55.705,-179.987,7.731,149.459
C03457=1120.629,80.753,-55.687,-179.988,7.727,149.458
C03458=1120.634,80.504,-55.669,-179.989,7.724,149.458
C03459=1120.639,80.254,-55.652,-179.990,7.720,149.457
C03460=1120.644,80.005,-55.634,-179.991,7.716,149.457
C03461=1120.649,79.756,-55.616,-179.992,7.712,149.456
C03462=1120.654,79.506,-55.598,-179.993,7.708,149.455
C03463=1120.658,79.257,-55.582,-179.995,7.704,149.455
C03464=1120.663,79.008,-55.564,-179.995,7.701,149.454
C03465=1120.668,78.759,-55.546,-179.997,7.697,149.454
C03466=1120.673,78.509,-55.528,-179.997,7.694,149.453
C03467=1120.678,78.260,-55.510,-179.999,7.690,149.453
C03468=1120.683,78.010,-55.492,-179.999,7.686,149.452
C03469=1120.688,77.761,-55.474,180.000,7.683,149.452
C03470=1120.692,77.512,-55.458,179.999,7.679,149.451
C03471=1120.697,77.263,-55.440,179.998,7.675,149.450
C03472=1120.702,77.013,-55.422,179.997,7.671,149.450
C03473=1120.707,76.764,-55.405,179.996,7.668,149.449
C03474=1120.712,76.549,-55.389,179.995,7.664,149.449
C03475=1120.716,76.335,-55.374,179.994,7.661,149.448
C03476=1120.720,76.120,-55.359,179.993,7.658,149.448
C03477=1120.724,75.906,-55.344,179.991,7.654,149.448
C03478=1120.728,75.691,-55.329,179.990,7.651,149.447
C03479=1120.733,75.477,-55.314,179.988,7.647,149.447
C03480=1120.737,75.262,-55.298,179.987,7.644,149.446
C03481=1120.741,75.047,-55.284,179.986,7.641,149.446
C03482=1120.745,74.798,-55.266,179.985,7.637,149.446
C03483=1120.750,74.549,-55.248,179.983,7.633,149.445
C03484=1120.756,74.299,-55.231,179.982,7.629,149.445
C03485=1120.760,74.050,-55.213,179.980,7.625,149.444
C03486=1120.765,73.800,-55.196,179.979,7.621,149.443
C03487=1120.770,73.551,-55.178,179.978,7.617,149.443
C03488=1120.776,73.302,-55.161,179.976,7.613,149.443
C03489=1120.781,73.053,-55.143,179.974,7.609,149.442
C03490=1120.785,72.803,-55.127,179.973,7.605,149.442
C03491=1120.790,72.554,-55.109,179.972,7.601,149.441
C03492=1120.795,72.304,-55.091,179.970,7.597,149.441
C03493=1120.799,72.056,-55.074,179.969,7.593,149.440
C03494=1120.805,71.806,-55.057,179.967,7.589,149.440
C03495=1120.810,71.556,-55.040,179.966,7.585,149.439
C03496=1120.814,71.307,-55.022,179.964,7.581,149.439
C03497=1120.819,71.057,-55.005,179.963,7.577,149.438
C03498=1120.825,70.809,-54.987,179.962,7.573,149.438
C03499=1120.829,70.559,-54.971,179.961,7.570,149.437
C03500=1120.834,70.310,-54.953,179.959,7.566,149.437
C03501=1120.839,70.061,-54.936,179.958,7.561,149.436
C03502=1120.844,69.811,-54.919,179.956,7.558,149.436
C03503=1120.849,69.561,-54.901,179.955,7.554,149.435
C03504=1120.853,69.312,-54.884,179.954,7.549,149.435
C03505=1120.859,69.063,-54.867,179.952,7.545,149.434
C03506=1120.863,68.814,-54.850,179.951,7.542,149.434
C03507=1120.868,68.565,-54.833,179.949,7.538,149.433
C03508=1120.874,68.315,-54.815,179.948,7.533,149.433
C03509=1120.878,68.065,-54.799,179.946,7.529,149.432
C03510=1120.883,67.815,-54.781,179.945,7.526,149.432
C03511=1120.888,67.567,-54.764,179.944,7.521,149.431
C03512=1120.893,67.317,-54.747,179.942,7.517,149.431
C03513=1120.898,67.068,-54.730,179.940,7.513,149.430
C03514=1120.903,66.818,-54.713,179.940,7.510,149.430
C03515=1120.907,66.569,-54.696,179.938,7.506,149.429
C03516=1120.913,66.320,-54.679,179.937,7.502,149.429
C03517=1120.917,66.071,-54.662,179.936,7.498,149.428
C03518=1120.923,65.821,-54.645,179.934,7.494,149.428
C03519=1120.927,65.571,-54.628,179.933,7.490,149.427
C03520=1120.933,65.322,-54.611,179.932,7.486,149.427
C03521=1120.937,65.074,-54.594,179.930,7.482,149.426
C03522=1120.942,64.824,-54.577,179.928,7.478,149.426
C03523=1120.947,64.574,-54.560,179.927,7.474,149.425
C03524=1120.951,64.325,-54.543,179.926,7.470,149.425
C03525=1120.957,64.076,-54.526,179.924,7.466,149.424
C03526=1120.962,63.826,-54.510,179.923,7.461,149.424
C03527=1120.967,63.576,-54.492,179.922,7.458,149.423
C03528=1120.972,63.328,-54.476,179.921,7.454,149.423
C03529=1120.977,63.078,-54.459,179.919,7.450,149.422
C03530=1120.981,62.863,-54.444,179.918,7.446,149.422
C03531=1120.986,62.649,-54.430,179.917,7.443,149.421
C03532=1120.989,62.434,-54.416,179.916,7.440,149.421
C03533=1120.994,62.220,-54.401,179.914,7.436,149.420
C03534=1120.998,62.005,-54.387,179.913,7.433,149.420
C03535=1121.002,61.791,-54.372,179.912,7.429,149.420
C03536=1121.006,61.576,-54.358,179.911,7.426,149.419
C03537=1121.011,61.361,-54.343,179.910,7.423,149.419
C03538=1121.016,61.111,-54.327,179.909,7.419,149.418
C03539=1121.020,60.862,-54.310,179.907,7.415,149.418
C03540=1121.025,60.612,-54.293,179.906,7.410,149.417
C03541=1121.030,60.363,-54.276,179.905,7.406,149.417
C03542=1121.035,60.114,-54.260,179.903,7.403,149.416
C03543=1121.041,59.865,-54.243,179.902,7.398,149.416
C03544=1121.045,59.615,-54.226,179.900,7.394,149.415
C03545=1121.050,59.366,-54.209,179.899,7.390,149.414
C03546=1121.055,59.116,-54.194,179.898,7.386,149.414
C03547=1121.060,58.867,-54.177,179.896,7.382,149.414
C03548=1121.065,58.617,-54.160,179.896,7.379,149.413
C03549=1121.070,58.368,-54.144,179.894,7.375,149.413
C03550=1121.075,58.119,-54.126,179.893,7.370,149.412
C03551=1121.080,57.869,-54.110,179.892,7.367,149.411
C03552=1121.085,57.620,-54.093,179.890,7.362,149.411
C03553=1121.089,57.370,-54.077,179.889,7.358,149.410
C03554=1121.095,57.121,-54.061,179.888,7.354,149.410
C03555=1121.100,56.872,-54.044,179.886,7.350,149.409
C03556=1121.104,56.622,-54.027,179.885,7.346,149.409
C03557=1121.109,56.373,-54.011,179.884,7.342,149.408
C03558=1121.114,56.123,-53.995,179.882,7.338,149.408
C03559=1121.120,55.874,-53.978,179.881,7.334,149.407
C03560=1121.124,55.625,-53.961,179.880,7.331,149.407
C03561=1121.130,55.375,-53.946,179.879,7.326,149.406
C03562=1121.134,55.126,-53.929,179.877,7.322,149.406
C03563=1121.139,54.876,-53.912,179.876,7.318,149.405
C03564=1121.144,54.627,-53.896,179.875,7.314,149.405
C03565=1121.149,54.377,-53.880,179.874,7.310,149.404
C03566=1121.154,54.128,-53.863,179.872,7.306,149.403
C03567=1121.159,53.879,-53.847,179.871,7.302,149.403
C03568=1121.164,53.629,-53.831,179.869,7.298,149.402
C03569=1121.169,53.380,-53.814,179.868,7.293,149.402
C03570=1121.174,53.131,-53.799,179.867,7.290,149.401
C03571=1121.179,52.881,-53.782,179.866,7.285,149.401
C03572=1121.184,52.632,-53.765,179.865,7.282,149.400
C03573=1121.189,52.382,-53.749,179.864,7.278,149.400
C03574=1121.194,52.133,-53.733,179.862,7.274,149.399
C03575=1121.199,51.883,-53.717,179.861,7.270,149.399
C03576=1121.204,51.634,-53.701,179.859,7.266,149.398
C03577=1121.209,51.385,-53.684,179.858,7.261,149.397
C03578=1121.214,51.135,-53.668,179.857,7.257,149.397
C03579=1121.218,50.886,-53.652,179.856,7.253,149.396
C03580=1121.224,50.636,-53.636,179.855,7.249,149.396
C03581=1121.228,50.387,-53.620,179.853,7.245,149.395
C03582=1121.234,50.138,-53.604,179.852,7.241,149.395
C03583=1121.238,49.888,-53.587,179.850,7.237,149.394
C03584=1121.244,49.639,-53.572,179.849,7.232,149.394
C03585=1121.248,49.389,-53.555,179.849,7.229,149.393
C03586=1121.253,49.174,-53.542,179.847,7.225,149.393
C03587=1121.258,48.960,-53.528,179.846,7.222,149.392
C03588=1121.261,48.745,-53.514,179.845,7.218,149.392
C03589=1121.266,48.530,-53.500,179.844,7.215,149.391
C03590=1121.270,48.316,-53.486,179.843,7.211,149.391
C03591=1121.274,48.101,-53.472,179.842,7.207,149.390
C03592=1121.278,47.886,-53.459,179.841,7.204,149.390
C03593=1121.283,47.671,-53.445,179.840,7.201,149.389
C03594=1121.288,47.422,-53.428,179.839,7.197,149.389
C03595=1121.292,47.173,-53.413,179.838,7.193,149.388
C03596=1121.297,46.923,-53.397,179.836,7.189,149.388
C03597=1121.302,46.674,-53.381,179.835,7.184,149.387
C03598=1121.308,46.424,-53.365,179.834,7.180,149.386
C03599=1121.312,46.174,-53.349,179.833,7.176,149.386
C03600=1121.318,45.926,-53.333,179.831,7.172,149.385
C03601=1121.322,45.675,-53.317,179.830,7.168,149.385
C03602=1121.328,45.426,-53.302,179.829,7.164,149.384
C03603=1121.333,45.177,-53.285,179.828,7.159,149.383
C03604=1121.338,44.927,-53.269,179.827,7.155,149.383
C03605=1121.342,44.678,-53.254,179.825,7.151,149.382
C03606=1121.348,44.429,-53.239,179.825,7.148,149.382
C03607=1121.352,44.179,-53.222,179.824,7.143,149.381
C03608=1121.358,43.930,-53.206,179.822,7.139,149.381
C03609=1121.362,43.680,-53.191,179.821,7.135,149.380
C03610=1121.368,43.430,-53.175,179.820,7.131,149.379
C03611=1121.372,43.181,-53.160,179.818,7.127,149.379
C03612=1121.377,42.932,-53.143,179.817,7.123,149.378
C03613=1121.382,42.682,-53.128,179.816,7.118,149.378
C03614=1121.388,42.433,-53.112,179.815,7.114,149.377
C03615=1121.392,42.183,-53.096,179.814,7.110,149.377
C03616=1121.397,41.934,-53.081,179.813,7.106,149.376
C03617=1121.402,41.685,-53.065,179.811,7.101,149.375
C03618=1121.407,41.436,-53.049,179.810,7.097,149.375
C03619=1121.412,41.185,-53.033,179.809,7.093,149.374
C03620=1121.418,40.936,-53.018,179.808,7.090,149.374
C03621=1121.422,40.687,-53.003,179.807,7.085,149.373
C03622=1121.427,40.437,-52.987,179.806,7.081,149.372
C03623=1121.432,40.187,-52.971,179.805,7.077,149.372
C03624=1121.438,39.938,-52.956,179.804,7.073,149.371
C03625=1121.443,39.689,-52.941,179.803,7.068,149.371
C03626=1121.447,39.439,-52.925,179.801,7.064,149.370
C03627=1121.453,39.189,-52.909,179.800,7.060,149.369
C03628=1121.457,38.940,-52.894,179.799,7.056,149.369
C03629=1121.463,38.691,-52.878,179.798,7.052,149.368
C03630=1121.468,38.441,-52.863,179.797,7.047,149.367
C03631=1121.472,38.192,-52.848,179.796,7.043,149.367
C03632=1121.478,37.942,-52.832,179.795,7.039,149.366
